ABB RAPID module: zignalmeister_2000.mod

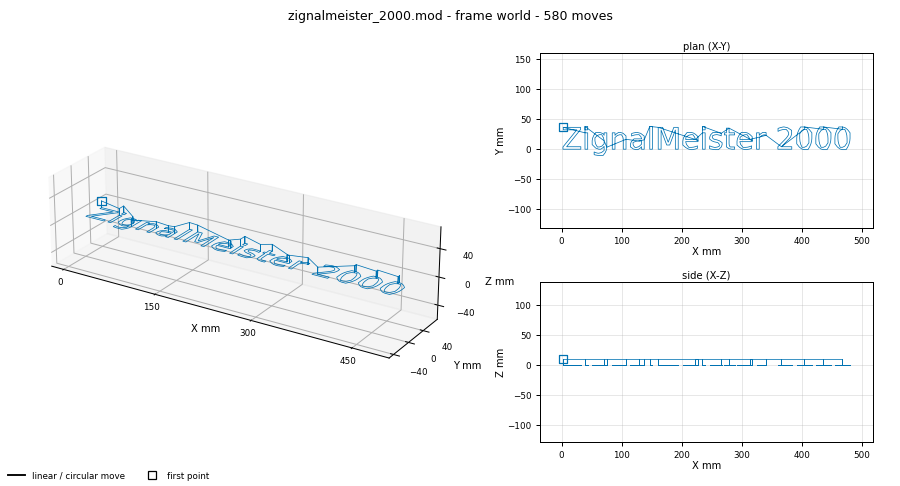
[picture p0: tool path of zignalmeister_2000.mod in frame world, 580 of 580 moves have a stored position in this frame; points joined in program order, loops and branches not executed]
MODULE TextDrawing
    ! Generated RAPID code for drawing text: ZignalMeister 2000
    ! Font: DejaVuSans.ttf
    ! Text size: 50.0 mm
    ! Point density: 5.0 mm
    ! Total points: 528
    ! Estimated time: 79.2 seconds

    ! Define target positions
    ! Path 1/26
    CONST robtarget p0:=[[2.81,36.45,0],[0,0,1,0],[-1,0,-1,0],[9E9,9E9,9E9,9E9,9E9,9E9]];
    CONST robtarget p1:=[[31.45,36.45,0],[0,0,1,0],[-1,0,-1,0],[9E9,9E9,9E9,9E9,9E9,9E9]];
    CONST robtarget p2:=[[31.45,32.69,0],[0,0,1,0],[-1,0,-1,0],[9E9,9E9,9E9,9E9,9E9,9E9]];
    CONST robtarget p3:=[[8.40,4.15,0],[0,0,1,0],[-1,0,-1,0],[9E9,9E9,9E9,9E9,9E9,9E9]];
    CONST robtarget p4:=[[32.01,4.15,0],[0,0,1,0],[-1,0,-1,0],[9E9,9E9,9E9,9E9,9E9,9E9]];
    CONST robtarget p5:=[[32.01,0.00,0],[0,0,1,0],[-1,0,-1,0],[9E9,9E9,9E9,9E9,9E9,9E9]];
    CONST robtarget p6:=[[2.25,0.00,0],[0,0,1,0],[-1,0,-1,0],[9E9,9E9,9E9,9E9,9E9,9E9]];
    CONST robtarget p7:=[[2.25,3.76,0],[0,0,1,0],[-1,0,-1,0],[9E9,9E9,9E9,9E9,9E9,9E9]];
    CONST robtarget p8:=[[25.29,32.30,0],[0,0,1,0],[-1,0,-1,0],[9E9,9E9,9E9,9E9,9E9,9E9]];
    CONST robtarget p9:=[[2.81,32.30,0],[0,0,1,0],[-1,0,-1,0],[9E9,9E9,9E9,9E9,9E9,9E9]];
    CONST robtarget p10:=[[2.81,36.45,0],[0,0,1,0],[-1,0,-1,0],[9E9,9E9,9E9,9E9,9E9,9E9]];
    ! Path 2/26
    CONST robtarget p11:=[[38.96,27.34,0],[0,0,1,0],[-1,0,-1,0],[9E9,9E9,9E9,9E9,9E9,9E9]];
    CONST robtarget p12:=[[43.46,27.34,0],[0,0,1,0],[-1,0,-1,0],[9E9,9E9,9E9,9E9,9E9,9E9]];
    CONST robtarget p13:=[[43.46,0.00,0],[0,0,1,0],[-1,0,-1,0],[9E9,9E9,9E9,9E9,9E9,9E9]];
    CONST robtarget p14:=[[38.96,0.00,0],[0,0,1,0],[-1,0,-1,0],[9E9,9E9,9E9,9E9,9E9,9E9]];
    CONST robtarget p15:=[[38.96,27.34,0],[0,0,1,0],[-1,0,-1,0],[9E9,9E9,9E9,9E9,9E9,9E9]];
    ! Path 3/26
    CONST robtarget p16:=[[38.96,37.99,0],[0,0,1,0],[-1,0,-1,0],[9E9,9E9,9E9,9E9,9E9,9E9]];
    CONST robtarget p17:=[[43.46,37.99,0],[0,0,1,0],[-1,0,-1,0],[9E9,9E9,9E9,9E9,9E9,9E9]];
    CONST robtarget p18:=[[43.46,32.30,0],[0,0,1,0],[-1,0,-1,0],[9E9,9E9,9E9,9E9,9E9,9E9]];
    CONST robtarget p19:=[[38.96,32.30,0],[0,0,1,0],[-1,0,-1,0],[9E9,9E9,9E9,9E9,9E9,9E9]];
    CONST robtarget p20:=[[38.96,37.99,0],[0,0,1,0],[-1,0,-1,0],[9E9,9E9,9E9,9E9,9E9,9E9]];
    ! Path 4/26
    CONST robtarget p21:=[[70.85,13.99,0],[0,0,1,0],[-1,0,-1,0],[9E9,9E9,9E9,9E9,9E9,9E9]];
    CONST robtarget p22:=[[69.84,18.99,0],[0,0,1,0],[-1,0,-1,0],[9E9,9E9,9E9,9E9,9E9,9E9]];
    CONST robtarget p23:=[[66.82,24.24,0],[0,0,1,0],[-1,0,-1,0],[9E9,9E9,9E9,9E9,9E9,9E9]];
    CONST robtarget p24:=[[65.91,24.24,0],[0,0,1,0],[-1,0,-1,0],[9E9,9E9,9E9,9E9,9E9,9E9]];
    CONST robtarget p25:=[[63.18,24.24,0],[0,0,1,0],[-1,0,-1,0],[9E9,9E9,9E9,9E9,9E9,9E9]];
    CONST robtarget p26:=[[59.47,22.90,0],[0,0,1,0],[-1,0,-1,0],[9E9,9E9,9E9,9E9,9E9,9E9]];
    CONST robtarget p27:=[[55.54,18.87,0],[0,0,1,0],[-1,0,-1,0],[9E9,9E9,9E9,9E9,9E9,9E9]];
    CONST robtarget p28:=[[55.54,17.65,0],[0,0,1,0],[-1,0,-1,0],[9E9,9E9,9E9,9E9,9E9,9E9]];
    CONST robtarget p29:=[[55.54,13.99,0],[0,0,1,0],[-1,0,-1,0],[9E9,9E9,9E9,9E9,9E9,9E9]];
    CONST robtarget p30:=[[56.55,9.00,0],[0,0,1,0],[-1,0,-1,0],[9E9,9E9,9E9,9E9,9E9,9E9]];
    CONST robtarget p31:=[[59.57,3.76,0],[0,0,1,0],[-1,0,-1,0],[9E9,9E9,9E9,9E9,9E9,9E9]];
    CONST robtarget p32:=[[60.47,3.76,0],[0,0,1,0],[-1,0,-1,0],[9E9,9E9,9E9,9E9,9E9,9E9]];
    CONST robtarget p33:=[[63.18,3.76,0],[0,0,1,0],[-1,0,-1,0],[9E9,9E9,9E9,9E9,9E9,9E9]];
    CONST robtarget p34:=[[66.92,5.10,0],[0,0,1,0],[-1,0,-1,0],[9E9,9E9,9E9,9E9,9E9,9E9]];
    CONST robtarget p35:=[[70.85,9.13,0],[0,0,1,0],[-1,0,-1,0],[9E9,9E9,9E9,9E9,9E9,9E9]];
    CONST robtarget p36:=[[70.85,10.35,0],[0,0,1,0],[-1,0,-1,0],[9E9,9E9,9E9,9E9,9E9,9E9]];
    CONST robtarget p37:=[[70.85,13.99,0],[0,0,1,0],[-1,0,-1,0],[9E9,9E9,9E9,9E9,9E9,9E9]];
    ! Path 5/26
    CONST robtarget p38:=[[75.34,3.39,0],[0,0,1,0],[-1,0,-1,0],[9E9,9E9,9E9,9E9,9E9,9E9]];
    CONST robtarget p39:=[[74.65,-1.24,0],[0,0,1,0],[-1,0,-1,0],[9E9,9E9,9E9,9E9,9E9,9E9]];
    CONST robtarget p40:=[[72.59,-5.84,0],[0,0,1,0],[-1,0,-1,0],[9E9,9E9,9E9,9E9,9E9,9E9]];
    CONST robtarget p41:=[[69.14,-10.40,0],[0,0,1,0],[-1,0,-1,0],[9E9,9E9,9E9,9E9,9E9,9E9]];
    CONST robtarget p42:=[[67.54,-10.40,0],[0,0,1,0],[-1,0,-1,0],[9E9,9E9,9E9,9E9,9E9,9E9]];
    CONST robtarget p43:=[[62.74,-10.40,0],[0,0,1,0],[-1,0,-1,0],[9E9,9E9,9E9,9E9,9E9,9E9]];
    CONST robtarget p44:=[[59.92,-10.22,0],[0,0,1,0],[-1,0,-1,0],[9E9,9E9,9E9,9E9,9E9,9E9]];
    CONST robtarget p45:=[[56.18,-9.69,0],[0,0,1,0],[-1,0,-1,0],[9E9,9E9,9E9,9E9,9E9,9E9]];
    CONST robtarget p46:=[[55.68,-9.51,0],[0,0,1,0],[-1,0,-1,0],[9E9,9E9,9E9,9E9,9E9,9E9]];
    CONST robtarget p47:=[[54.20,-8.96,0],[0,0,1,0],[-1,0,-1,0],[9E9,9E9,9E9,9E9,9E9,9E9]];
    CONST robtarget p48:=[[54.20,-4.59,0],[0,0,1,0],[-1,0,-1,0],[9E9,9E9,9E9,9E9,9E9,9E9]];
    CONST robtarget p49:=[[56.65,-5.65,0],[0,0,1,0],[-1,0,-1,0],[9E9,9E9,9E9,9E9,9E9,9E9]];
    CONST robtarget p50:=[[60.03,-6.69,0],[0,0,1,0],[-1,0,-1,0],[9E9,9E9,9E9,9E9,9E9,9E9]];
    CONST robtarget p51:=[[60.53,-6.69,0],[0,0,1,0],[-1,0,-1,0],[9E9,9E9,9E9,9E9,9E9,9E9]];
    CONST robtarget p52:=[[62.04,-6.69,0],[0,0,1,0],[-1,0,-1,0],[9E9,9E9,9E9,9E9,9E9,9E9]];
    CONST robtarget p53:=[[66.45,-5.54,0],[0,0,1,0],[-1,0,-1,0],[9E9,9E9,9E9,9E9,9E9,9E9]];
    CONST robtarget p54:=[[70.85,-2.08,0],[0,0,1,0],[-1,0,-1,0],[9E9,9E9,9E9,9E9,9E9,9E9]];
    CONST robtarget p55:=[[70.85,-0.91,0],[0,0,1,0],[-1,0,-1,0],[9E9,9E9,9E9,9E9,9E9,9E9]];
    CONST robtarget p56:=[[70.85,2.59,0],[0,0,1,0],[-1,0,-1,0],[9E9,9E9,9E9,9E9,9E9,9E9]];
    CONST robtarget p57:=[[70.85,4.81,0],[0,0,1,0],[-1,0,-1,0],[9E9,9E9,9E9,9E9,9E9,9E9]];
    CONST robtarget p58:=[[68.72,2.40,0],[0,0,1,0],[-1,0,-1,0],[9E9,9E9,9E9,9E9,9E9,9E9]];
    CONST robtarget p59:=[[65.11,0.00,0],[0,0,1,0],[-1,0,-1,0],[9E9,9E9,9E9,9E9,9E9,9E9]];
    CONST robtarget p60:=[[64.36,0.00,0],[0,0,1,0],[-1,0,-1,0],[9E9,9E9,9E9,9E9,9E9,9E9]];
    CONST robtarget p61:=[[62.08,0.00,0],[0,0,1,0],[-1,0,-1,0],[9E9,9E9,9E9,9E9,9E9,9E9]];
    CONST robtarget p62:=[[56.77,1.92,0],[0,0,1,0],[-1,0,-1,0],[9E9,9E9,9E9,9E9,9E9,9E9]];
    CONST robtarget p63:=[[50.90,7.67,0],[0,0,1,0],[-1,0,-1,0],[9E9,9E9,9E9,9E9,9E9,9E9]];
    CONST robtarget p64:=[[50.90,9.25,0],[0,0,1,0],[-1,0,-1,0],[9E9,9E9,9E9,9E9,9E9,9E9]];
    CONST robtarget p65:=[[50.90,13.99,0],[0,0,1,0],[-1,0,-1,0],[9E9,9E9,9E9,9E9,9E9,9E9]];
    CONST robtarget p66:=[[51.59,18.37,0],[0,0,1,0],[-1,0,-1,0],[9E9,9E9,9E9,9E9,9E9,9E9]];
    CONST robtarget p67:=[[53.64,23.04,0],[0,0,1,0],[-1,0,-1,0],[9E9,9E9,9E9,9E9,9E9,9E9]];
    CONST robtarget p68:=[[57.06,28.00,0],[0,0,1,0],[-1,0,-1,0],[9E9,9E9,9E9,9E9,9E9,9E9]];
    CONST robtarget p69:=[[58.31,28.00,0],[0,0,1,0],[-1,0,-1,0],[9E9,9E9,9E9,9E9,9E9,9E9]];
    CONST robtarget p70:=[[62.08,28.00,0],[0,0,1,0],[-1,0,-1,0],[9E9,9E9,9E9,9E9,9E9,9E9]];
    CONST robtarget p71:=[[65.44,27.40,0],[0,0,1,0],[-1,0,-1,0],[9E9,9E9,9E9,9E9,9E9,9E9]];
    CONST robtarget p72:=[[69.46,25.61,0],[0,0,1,0],[-1,0,-1,0],[9E9,9E9,9E9,9E9,9E9,9E9]];
    CONST robtarget p73:=[[69.81,25.01,0],[0,0,1,0],[-1,0,-1,0],[9E9,9E9,9E9,9E9,9E9,9E9]];
    CONST robtarget p74:=[[70.85,23.19,0],[0,0,1,0],[-1,0,-1,0],[9E9,9E9,9E9,9E9,9E9,9E9]];
    CONST robtarget p75:=[[70.85,27.34,0],[0,0,1,0],[-1,0,-1,0],[9E9,9E9,9E9,9E9,9E9,9E9]];
    CONST robtarget p76:=[[75.34,27.34,0],[0,0,1,0],[-1,0,-1,0],[9E9,9E9,9E9,9E9,9E9,9E9]];
    CONST robtarget p77:=[[75.34,3.39,0],[0,0,1,0],[-1,0,-1,0],[9E9,9E9,9E9,9E9,9E9,9E9]];
    ! Path 6/26
    CONST robtarget p78:=[[107.32,16.50,0],[0,0,1,0],[-1,0,-1,0],[9E9,9E9,9E9,9E9,9E9,9E9]];
    CONST robtarget p79:=[[107.32,0.00,0],[0,0,1,0],[-1,0,-1,0],[9E9,9E9,9E9,9E9,9E9,9E9]];
    CONST robtarget p80:=[[102.83,0.00,0],[0,0,1,0],[-1,0,-1,0],[9E9,9E9,9E9,9E9,9E9,9E9]];
    CONST robtarget p81:=[[102.83,16.36,0],[0,0,1,0],[-1,0,-1,0],[9E9,9E9,9E9,9E9,9E9,9E9]];
    CONST robtarget p82:=[[102.08,20.23,0],[0,0,1,0],[-1,0,-1,0],[9E9,9E9,9E9,9E9,9E9,9E9]];
    CONST robtarget p83:=[[99.80,24.10,0],[0,0,1,0],[-1,0,-1,0],[9E9,9E9,9E9,9E9,9E9,9E9]];
    CONST robtarget p84:=[[99.05,24.10,0],[0,0,1,0],[-1,0,-1,0],[9E9,9E9,9E9,9E9,9E9,9E9]];
    CONST robtarget p85:=[[96.78,24.10,0],[0,0,1,0],[-1,0,-1,0],[9E9,9E9,9E9,9E9,9E9,9E9]];
    CONST robtarget p86:=[[93.00,22.94,0],[0,0,1,0],[-1,0,-1,0],[9E9,9E9,9E9,9E9,9E9,9E9]];
    CONST robtarget p87:=[[88.94,19.46,0],[0,0,1,0],[-1,0,-1,0],[9E9,9E9,9E9,9E9,9E9,9E9]];
    CONST robtarget p88:=[[88.94,18.46,0],[0,0,1,0],[-1,0,-1,0],[9E9,9E9,9E9,9E9,9E9,9E9]];
    CONST robtarget p89:=[[88.94,15.45,0],[0,0,1,0],[-1,0,-1,0],[9E9,9E9,9E9,9E9,9E9,9E9]];
    CONST robtarget p90:=[[88.94,0.00,0],[0,0,1,0],[-1,0,-1,0],[9E9,9E9,9E9,9E9,9E9,9E9]];
    CONST robtarget p91:=[[84.42,0.00,0],[0,0,1,0],[-1,0,-1,0],[9E9,9E9,9E9,9E9,9E9,9E9]];
    CONST robtarget p92:=[[84.42,27.34,0],[0,0,1,0],[-1,0,-1,0],[9E9,9E9,9E9,9E9,9E9,9E9]];
    CONST robtarget p93:=[[88.94,27.34,0],[0,0,1,0],[-1,0,-1,0],[9E9,9E9,9E9,9E9,9E9,9E9]];
    CONST robtarget p94:=[[88.94,23.10,0],[0,0,1,0],[-1,0,-1,0],[9E9,9E9,9E9,9E9,9E9,9E9]];
    CONST robtarget p95:=[[91.24,25.56,0],[0,0,1,0],[-1,0,-1,0],[9E9,9E9,9E9,9E9,9E9,9E9]];
    CONST robtarget p96:=[[94.92,28.00,0],[0,0,1,0],[-1,0,-1,0],[9E9,9E9,9E9,9E9,9E9,9E9]];
    CONST robtarget p97:=[[95.64,28.00,0],[0,0,1,0],[-1,0,-1,0],[9E9,9E9,9E9,9E9,9E9,9E9]];
    CONST robtarget p98:=[[97.78,28.00,0],[0,0,1,0],[-1,0,-1,0],[9E9,9E9,9E9,9E9,9E9,9E9]];
    CONST robtarget p99:=[[102.52,26.54,0],[0,0,1,0],[-1,0,-1,0],[9E9,9E9,9E9,9E9,9E9,9E9]];
    CONST robtarget p100:=[[107.32,22.17,0],[0,0,1,0],[-1,0,-1,0],[9E9,9E9,9E9,9E9,9E9,9E9]];
    CONST robtarget p101:=[[107.32,20.75,0],[0,0,1,0],[-1,0,-1,0],[9E9,9E9,9E9,9E9,9E9,9E9]];
    CONST robtarget p102:=[[107.32,16.50,0],[0,0,1,0],[-1,0,-1,0],[9E9,9E9,9E9,9E9,9E9,9E9]];
    ! Path 7/26
    CONST robtarget p103:=[[128.71,13.75,0],[0,0,1,0],[-1,0,-1,0],[9E9,9E9,9E9,9E9,9E9,9E9]];
    CONST robtarget p104:=[[123.58,13.12,0],[0,0,1,0],[-1,0,-1,0],[9E9,9E9,9E9,9E9,9E9,9E9]];
    CONST robtarget p105:=[[119.07,11.25,0],[0,0,1,0],[-1,0,-1,0],[9E9,9E9,9E9,9E9,9E9,9E9]];
    CONST robtarget p106:=[[119.07,10.50,0],[0,0,1,0],[-1,0,-1,0],[9E9,9E9,9E9,9E9,9E9,9E9]];
    CONST robtarget p107:=[[119.07,8.25,0],[0,0,1,0],[-1,0,-1,0],[9E9,9E9,9E9,9E9,9E9,9E9]];
    CONST robtarget p108:=[[119.85,5.76,0],[0,0,1,0],[-1,0,-1,0],[9E9,9E9,9E9,9E9,9E9,9E9]];
    CONST robtarget p109:=[[122.22,3.05,0],[0,0,1,0],[-1,0,-1,0],[9E9,9E9,9E9,9E9,9E9,9E9]];
    CONST robtarget p110:=[[122.89,3.05,0],[0,0,1,0],[-1,0,-1,0],[9E9,9E9,9E9,9E9,9E9,9E9]];
    CONST robtarget p111:=[[124.93,3.05,0],[0,0,1,0],[-1,0,-1,0],[9E9,9E9,9E9,9E9,9E9,9E9]];
    CONST robtarget p112:=[[128.86,4.38,0],[0,0,1,0],[-1,0,-1,0],[9E9,9E9,9E9,9E9,9E9,9E9]];
    CONST robtarget p113:=[[133.18,8.35,0],[0,0,1,0],[-1,0,-1,0],[9E9,9E9,9E9,9E9,9E9,9E9]];
    CONST robtarget p114:=[[133.18,9.45,0],[0,0,1,0],[-1,0,-1,0],[9E9,9E9,9E9,9E9,9E9,9E9]];
    CONST robtarget p115:=[[133.18,12.74,0],[0,0,1,0],[-1,0,-1,0],[9E9,9E9,9E9,9E9,9E9,9E9]];
    CONST robtarget p116:=[[133.18,13.75,0],[0,0,1,0],[-1,0,-1,0],[9E9,9E9,9E9,9E9,9E9,9E9]];
    CONST robtarget p117:=[[128.71,13.75,0],[0,0,1,0],[-1,0,-1,0],[9E9,9E9,9E9,9E9,9E9,9E9]];
    ! Path 8/26
    CONST robtarget p118:=[[137.67,15.60,0],[0,0,1,0],[-1,0,-1,0],[9E9,9E9,9E9,9E9,9E9,9E9]];
    CONST robtarget p119:=[[137.67,0.00,0],[0,0,1,0],[-1,0,-1,0],[9E9,9E9,9E9,9E9,9E9,9E9]];
    CONST robtarget p120:=[[133.18,0.00,0],[0,0,1,0],[-1,0,-1,0],[9E9,9E9,9E9,9E9,9E9,9E9]];
    CONST robtarget p121:=[[133.18,4.15,0],[0,0,1,0],[-1,0,-1,0],[9E9,9E9,9E9,9E9,9E9,9E9]];
    CONST robtarget p122:=[[130.88,1.69,0],[0,0,1,0],[-1,0,-1,0],[9E9,9E9,9E9,9E9,9E9,9E9]];
    CONST robtarget p123:=[[127.05,-0.71,0],[0,0,1,0],[-1,0,-1,0],[9E9,9E9,9E9,9E9,9E9,9E9]];
    CONST robtarget p124:=[[126.22,-0.71,0],[0,0,1,0],[-1,0,-1,0],[9E9,9E9,9E9,9E9,9E9,9E9]];
    CONST robtarget p125:=[[123.73,-0.71,0],[0,0,1,0],[-1,0,-1,0],[9E9,9E9,9E9,9E9,9E9,9E9]];
    CONST robtarget p126:=[[119.34,0.47,0],[0,0,1,0],[-1,0,-1,0],[9E9,9E9,9E9,9E9,9E9,9E9]];
    CONST robtarget p127:=[[114.58,4.00,0],[0,0,1,0],[-1,0,-1,0],[9E9,9E9,9E9,9E9,9E9,9E9]];
    CONST robtarget p128:=[[114.58,4.99,0],[0,0,1,0],[-1,0,-1,0],[9E9,9E9,9E9,9E9,9E9,9E9]];
    CONST robtarget p129:=[[114.58,7.96,0],[0,0,1,0],[-1,0,-1,0],[9E9,9E9,9E9,9E9,9E9,9E9]];
    CONST robtarget p130:=[[116.12,12.59,0],[0,0,1,0],[-1,0,-1,0],[9E9,9E9,9E9,9E9,9E9,9E9]];
    CONST robtarget p131:=[[120.75,17.26,0],[0,0,1,0],[-1,0,-1,0],[9E9,9E9,9E9,9E9,9E9,9E9]];
    CONST robtarget p132:=[[122.28,17.26,0],[0,0,1,0],[-1,0,-1,0],[9E9,9E9,9E9,9E9,9E9,9E9]];
    CONST robtarget p133:=[[126.88,17.26,0],[0,0,1,0],[-1,0,-1,0],[9E9,9E9,9E9,9E9,9E9,9E9]];
    CONST robtarget p134:=[[133.18,17.26,0],[0,0,1,0],[-1,0,-1,0],[9E9,9E9,9E9,9E9,9E9,9E9]];
    CONST robtarget p135:=[[133.18,17.70,0],[0,0,1,0],[-1,0,-1,0],[9E9,9E9,9E9,9E9,9E9,9E9]];
    CONST robtarget p136:=[[132.16,20.87,0],[0,0,1,0],[-1,0,-1,0],[9E9,9E9,9E9,9E9,9E9,9E9]];
    CONST robtarget p137:=[[129.10,24.19,0],[0,0,1,0],[-1,0,-1,0],[9E9,9E9,9E9,9E9,9E9,9E9]];
    CONST robtarget p138:=[[128.18,24.19,0],[0,0,1,0],[-1,0,-1,0],[9E9,9E9,9E9,9E9,9E9,9E9]];
    CONST robtarget p139:=[[125.42,24.19,0],[0,0,1,0],[-1,0,-1,0],[9E9,9E9,9E9,9E9,9E9,9E9]];
    CONST robtarget p140:=[[122.55,23.91,0],[0,0,1,0],[-1,0,-1,0],[9E9,9E9,9E9,9E9,9E9,9E9]];
    CONST robtarget p141:=[[118.63,23.07,0],[0,0,1,0],[-1,0,-1,0],[9E9,9E9,9E9,9E9,9E9,9E9]];
    CONST robtarget p142:=[[118.12,22.79,0],[0,0,1,0],[-1,0,-1,0],[9E9,9E9,9E9,9E9,9E9,9E9]];
    CONST robtarget p143:=[[116.58,21.95,0],[0,0,1,0],[-1,0,-1,0],[9E9,9E9,9E9,9E9,9E9,9E9]];
    CONST robtarget p144:=[[116.58,26.10,0],[0,0,1,0],[-1,0,-1,0],[9E9,9E9,9E9,9E9,9E9,9E9]];
    CONST robtarget p145:=[[119.59,27.05,0],[0,0,1,0],[-1,0,-1,0],[9E9,9E9,9E9,9E9,9E9,9E9]];
    CONST robtarget p146:=[[123.68,28.00,0],[0,0,1,0],[-1,0,-1,0],[9E9,9E9,9E9,9E9,9E9,9E9]];
    CONST robtarget p147:=[[124.23,28.00,0],[0,0,1,0],[-1,0,-1,0],[9E9,9E9,9E9,9E9,9E9,9E9]];
    CONST robtarget p148:=[[125.88,28.00,0],[0,0,1,0],[-1,0,-1,0],[9E9,9E9,9E9,9E9,9E9,9E9]];
    CONST robtarget p149:=[[131.79,26.46,0],[0,0,1,0],[-1,0,-1,0],[9E9,9E9,9E9,9E9,9E9,9E9]];
    CONST robtarget p150:=[[137.67,21.85,0],[0,0,1,0],[-1,0,-1,0],[9E9,9E9,9E9,9E9,9E9,9E9]];
    CONST robtarget p151:=[[137.67,20.29,0],[0,0,1,0],[-1,0,-1,0],[9E9,9E9,9E9,9E9,9E9,9E9]];
    CONST robtarget p152:=[[137.67,15.60,0],[0,0,1,0],[-1,0,-1,0],[9E9,9E9,9E9,9E9,9E9,9E9]];
    ! Path 9/26
    CONST robtarget p153:=[[146.92,37.99,0],[0,0,1,0],[-1,0,-1,0],[9E9,9E9,9E9,9E9,9E9,9E9]];
    CONST robtarget p154:=[[151.42,37.99,0],[0,0,1,0],[-1,0,-1,0],[9E9,9E9,9E9,9E9,9E9,9E9]];
    CONST robtarget p155:=[[151.42,0.00,0],[0,0,1,0],[-1,0,-1,0],[9E9,9E9,9E9,9E9,9E9,9E9]];
    CONST robtarget p156:=[[146.92,0.00,0],[0,0,1,0],[-1,0,-1,0],[9E9,9E9,9E9,9E9,9E9,9E9]];
    CONST robtarget p157:=[[146.92,37.99,0],[0,0,1,0],[-1,0,-1,0],[9E9,9E9,9E9,9E9,9E9,9E9]];
    ! Path 10/26
    CONST robtarget p158:=[[161.01,36.45,0],[0,0,1,0],[-1,0,-1,0],[9E9,9E9,9E9,9E9,9E9,9E9]];
    CONST robtarget p159:=[[168.36,36.45,0],[0,0,1,0],[-1,0,-1,0],[9E9,9E9,9E9,9E9,9E9,9E9]];
    CONST robtarget p160:=[[177.66,11.65,0],[0,0,1,0],[-1,0,-1,0],[9E9,9E9,9E9,9E9,9E9,9E9]];
    CONST robtarget p161:=[[187.01,36.45,0],[0,0,1,0],[-1,0,-1,0],[9E9,9E9,9E9,9E9,9E9,9E9]];
    CONST robtarget p162:=[[194.36,36.45,0],[0,0,1,0],[-1,0,-1,0],[9E9,9E9,9E9,9E9,9E9,9E9]];
    CONST robtarget p163:=[[194.36,0.00,0],[0,0,1,0],[-1,0,-1,0],[9E9,9E9,9E9,9E9,9E9,9E9]];
    CONST robtarget p164:=[[189.55,0.00,0],[0,0,1,0],[-1,0,-1,0],[9E9,9E9,9E9,9E9,9E9,9E9]];
    CONST robtarget p165:=[[189.55,32.01,0],[0,0,1,0],[-1,0,-1,0],[9E9,9E9,9E9,9E9,9E9,9E9]];
    CONST robtarget p166:=[[180.15,7.01,0],[0,0,1,0],[-1,0,-1,0],[9E9,9E9,9E9,9E9,9E9,9E9]];
    CONST robtarget p167:=[[175.20,7.01,0],[0,0,1,0],[-1,0,-1,0],[9E9,9E9,9E9,9E9,9E9,9E9]];
    CONST robtarget p168:=[[165.80,32.01,0],[0,0,1,0],[-1,0,-1,0],[9E9,9E9,9E9,9E9,9E9,9E9]];
    CONST robtarget p169:=[[165.80,0.00,0],[0,0,1,0],[-1,0,-1,0],[9E9,9E9,9E9,9E9,9E9,9E9]];
    CONST robtarget p170:=[[161.01,0.00,0],[0,0,1,0],[-1,0,-1,0],[9E9,9E9,9E9,9E9,9E9,9E9]];
    CONST robtarget p171:=[[161.01,36.45,0],[0,0,1,0],[-1,0,-1,0],[9E9,9E9,9E9,9E9,9E9,9E9]];
    ! Path 11/26
    CONST robtarget p172:=[[227.34,14.79,0],[0,0,1,0],[-1,0,-1,0],[9E9,9E9,9E9,9E9,9E9,9E9]];
    CONST robtarget p173:=[[227.34,12.60,0],[0,0,1,0],[-1,0,-1,0],[9E9,9E9,9E9,9E9,9E9,9E9]];
    CONST robtarget p174:=[[206.69,12.60,0],[0,0,1,0],[-1,0,-1,0],[9E9,9E9,9E9,9E9,9E9,9E9]];
    CONST robtarget p175:=[[208.16,7.90,0],[0,0,1,0],[-1,0,-1,0],[9E9,9E9,9E9,9E9,9E9,9E9]];
    CONST robtarget p176:=[[211.99,3.10,0],[0,0,1,0],[-1,0,-1,0],[9E9,9E9,9E9,9E9,9E9,9E9]];
    CONST robtarget p177:=[[213.10,3.10,0],[0,0,1,0],[-1,0,-1,0],[9E9,9E9,9E9,9E9,9E9,9E9]];
    CONST robtarget p178:=[[216.46,3.10,0],[0,0,1,0],[-1,0,-1,0],[9E9,9E9,9E9,9E9,9E9,9E9]];
    CONST robtarget p179:=[[219.61,3.42,0],[0,0,1,0],[-1,0,-1,0],[9E9,9E9,9E9,9E9,9E9,9E9]];
    CONST robtarget p180:=[[223.90,4.37,0],[0,0,1,0],[-1,0,-1,0],[9E9,9E9,9E9,9E9,9E9,9E9]];
    CONST robtarget p181:=[[224.50,4.69,0],[0,0,1,0],[-1,0,-1,0],[9E9,9E9,9E9,9E9,9E9,9E9]];
    CONST robtarget p182:=[[226.29,5.64,0],[0,0,1,0],[-1,0,-1,0],[9E9,9E9,9E9,9E9,9E9,9E9]];
    CONST robtarget p183:=[[226.29,1.39,0],[0,0,1,0],[-1,0,-1,0],[9E9,9E9,9E9,9E9,9E9,9E9]];
    CONST robtarget p184:=[[223.21,0.35,0],[0,0,1,0],[-1,0,-1,0],[9E9,9E9,9E9,9E9,9E9,9E9]];
    CONST robtarget p185:=[[218.80,-0.71,0],[0,0,1,0],[-1,0,-1,0],[9E9,9E9,9E9,9E9,9E9,9E9]];
    CONST robtarget p186:=[[218.15,-0.71,0],[0,0,1,0],[-1,0,-1,0],[9E9,9E9,9E9,9E9,9E9,9E9]];
    CONST robtarget p187:=[[216.19,-0.71,0],[0,0,1,0],[-1,0,-1,0],[9E9,9E9,9E9,9E9,9E9,9E9]];
    CONST robtarget p188:=[[211.70,0.14,0],[0,0,1,0],[-1,0,-1,0],[9E9,9E9,9E9,9E9,9E9,9E9]];
    CONST robtarget p189:=[[206.97,2.68,0],[0,0,1,0],[-1,0,-1,0],[9E9,9E9,9E9,9E9,9E9,9E9]];
    CONST robtarget p190:=[[202.00,6.91,0],[0,0,1,0],[-1,0,-1,0],[9E9,9E9,9E9,9E9,9E9,9E9]];
    CONST robtarget p191:=[[202.00,8.53,0],[0,0,1,0],[-1,0,-1,0],[9E9,9E9,9E9,9E9,9E9,9E9]];
    CONST robtarget p192:=[[202.00,13.40,0],[0,0,1,0],[-1,0,-1,0],[9E9,9E9,9E9,9E9,9E9,9E9]];
    CONST robtarget p193:=[[202.81,18.01,0],[0,0,1,0],[-1,0,-1,0],[9E9,9E9,9E9,9E9,9E9,9E9]];
    CONST robtarget p194:=[[205.22,22.88,0],[0,0,1,0],[-1,0,-1,0],[9E9,9E9,9E9,9E9,9E9,9E9]];
    CONST robtarget p195:=[[209.25,28.00,0],[0,0,1,0],[-1,0,-1,0],[9E9,9E9,9E9,9E9,9E9,9E9]];
    CONST robtarget p196:=[[210.79,28.00,0],[0,0,1,0],[-1,0,-1,0],[9E9,9E9,9E9,9E9,9E9,9E9]];
    CONST robtarget p197:=[[215.41,28.00,0],[0,0,1,0],[-1,0,-1,0],[9E9,9E9,9E9,9E9,9E9,9E9]];
    CONST robtarget p198:=[[219.18,27.21,0],[0,0,1,0],[-1,0,-1,0],[9E9,9E9,9E9,9E9,9E9,9E9]];
    CONST robtarget p199:=[[223.16,24.85,0],[0,0,1,0],[-1,0,-1,0],[9E9,9E9,9E9,9E9,9E9,9E9]];
    CONST robtarget p200:=[[227.34,20.90,0],[0,0,1,0],[-1,0,-1,0],[9E9,9E9,9E9,9E9,9E9,9E9]];
    CONST robtarget p201:=[[227.34,19.37,0],[0,0,1,0],[-1,0,-1,0],[9E9,9E9,9E9,9E9,9E9,9E9]];
    CONST robtarget p202:=[[227.34,14.79,0],[0,0,1,0],[-1,0,-1,0],[9E9,9E9,9E9,9E9,9E9,9E9]];
    ! Path 12/26
    CONST robtarget p203:=[[222.85,16.11,0],[0,0,1,0],[-1,0,-1,0],[9E9,9E9,9E9,9E9,9E9,9E9]];
    CONST robtarget p204:=[[221.81,19.98,0],[0,0,1,0],[-1,0,-1,0],[9E9,9E9,9E9,9E9,9E9,9E9]];
    CONST robtarget p205:=[[218.77,24.19,0],[0,0,1,0],[-1,0,-1,0],[9E9,9E9,9E9,9E9,9E9,9E9]];
    CONST robtarget p206:=[[217.94,24.19,0],[0,0,1,0],[-1,0,-1,0],[9E9,9E9,9E9,9E9,9E9,9E9]];
    CONST robtarget p207:=[[215.45,24.19,0],[0,0,1,0],[-1,0,-1,0],[9E9,9E9,9E9,9E9,9E9,9E9]];
    CONST robtarget p208:=[[211.51,23.13,0],[0,0,1,0],[-1,0,-1,0],[9E9,9E9,9E9,9E9,9E9,9E9]];
    CONST robtarget p209:=[[207.18,19.95,0],[0,0,1,0],[-1,0,-1,0],[9E9,9E9,9E9,9E9,9E9,9E9]];
    CONST robtarget p210:=[[207.09,18.98,0],[0,0,1,0],[-1,0,-1,0],[9E9,9E9,9E9,9E9,9E9,9E9]];
    CONST robtarget p211:=[[206.84,16.09,0],[0,0,1,0],[-1,0,-1,0],[9E9,9E9,9E9,9E9,9E9,9E9]];
    CONST robtarget p212:=[[222.85,16.11,0],[0,0,1,0],[-1,0,-1,0],[9E9,9E9,9E9,9E9,9E9,9E9]];
    ! Path 13/26
    CONST robtarget p213:=[[234.72,27.34,0],[0,0,1,0],[-1,0,-1,0],[9E9,9E9,9E9,9E9,9E9,9E9]];
    CONST robtarget p214:=[[239.21,27.34,0],[0,0,1,0],[-1,0,-1,0],[9E9,9E9,9E9,9E9,9E9,9E9]];
    CONST robtarget p215:=[[239.21,0.00,0],[0,0,1,0],[-1,0,-1,0],[9E9,9E9,9E9,9E9,9E9,9E9]];
    CONST robtarget p216:=[[234.72,0.00,0],[0,0,1,0],[-1,0,-1,0],[9E9,9E9,9E9,9E9,9E9,9E9]];
    CONST robtarget p217:=[[234.72,27.34,0],[0,0,1,0],[-1,0,-1,0],[9E9,9E9,9E9,9E9,9E9,9E9]];
    ! Path 14/26
    CONST robtarget p218:=[[234.72,37.99,0],[0,0,1,0],[-1,0,-1,0],[9E9,9E9,9E9,9E9,9E9,9E9]];
    CONST robtarget p219:=[[239.21,37.99,0],[0,0,1,0],[-1,0,-1,0],[9E9,9E9,9E9,9E9,9E9,9E9]];
    CONST robtarget p220:=[[239.21,32.30,0],[0,0,1,0],[-1,0,-1,0],[9E9,9E9,9E9,9E9,9E9,9E9]];
    CONST robtarget p221:=[[234.72,32.30,0],[0,0,1,0],[-1,0,-1,0],[9E9,9E9,9E9,9E9,9E9,9E9]];
    CONST robtarget p222:=[[234.72,37.99,0],[0,0,1,0],[-1,0,-1,0],[9E9,9E9,9E9,9E9,9E9,9E9]];
    ! Path 15/26
    CONST robtarget p223:=[[266.04,26.54,0],[0,0,1,0],[-1,0,-1,0],[9E9,9E9,9E9,9E9,9E9,9E9]];
    CONST robtarget p224:=[[266.04,22.29,0],[0,0,1,0],[-1,0,-1,0],[9E9,9E9,9E9,9E9,9E9,9E9]];
    CONST robtarget p225:=[[263.59,23.27,0],[0,0,1,0],[-1,0,-1,0],[9E9,9E9,9E9,9E9,9E9,9E9]];
    CONST robtarget p226:=[[260.03,24.24,0],[0,0,1,0],[-1,0,-1,0],[9E9,9E9,9E9,9E9,9E9,9E9]];
    CONST robtarget p227:=[[259.48,24.24,0],[0,0,1,0],[-1,0,-1,0],[9E9,9E9,9E9,9E9,9E9,9E9]];
    CONST robtarget p228:=[[257.84,24.24,0],[0,0,1,0],[-1,0,-1,0],[9E9,9E9,9E9,9E9,9E9,9E9]];
    CONST robtarget p229:=[[254.49,23.73,0],[0,0,1,0],[-1,0,-1,0],[9E9,9E9,9E9,9E9,9E9,9E9]];
    CONST robtarget p230:=[[251.15,22.19,0],[0,0,1,0],[-1,0,-1,0],[9E9,9E9,9E9,9E9,9E9,9E9]];
    CONST robtarget p231:=[[251.15,21.68,0],[0,0,1,0],[-1,0,-1,0],[9E9,9E9,9E9,9E9,9E9,9E9]];
    CONST robtarget p232:=[[251.15,20.14,0],[0,0,1,0],[-1,0,-1,0],[9E9,9E9,9E9,9E9,9E9,9E9]];
    CONST robtarget p233:=[[251.75,18.52,0],[0,0,1,0],[-1,0,-1,0],[9E9,9E9,9E9,9E9,9E9,9E9]];
    CONST robtarget p234:=[[253.54,16.80,0],[0,0,1,0],[-1,0,-1,0],[9E9,9E9,9E9,9E9,9E9,9E9]];
    CONST robtarget p235:=[[254.44,16.60,0],[0,0,1,0],[-1,0,-1,0],[9E9,9E9,9E9,9E9,9E9,9E9]];
    CONST robtarget p236:=[[257.15,15.99,0],[0,0,1,0],[-1,0,-1,0],[9E9,9E9,9E9,9E9,9E9,9E9]];
    CONST robtarget p237:=[[258.69,15.65,0],[0,0,1,0],[-1,0,-1,0],[9E9,9E9,9E9,9E9,9E9,9E9]];
    CONST robtarget p238:=[[263.29,13.95,0],[0,0,1,0],[-1,0,-1,0],[9E9,9E9,9E9,9E9,9E9,9E9]];
    CONST robtarget p239:=[[267.50,10.89,0],[0,0,1,0],[-1,0,-1,0],[9E9,9E9,9E9,9E9,9E9,9E9]];
    CONST robtarget p240:=[[267.50,10.05,0],[0,0,1,0],[-1,0,-1,0],[9E9,9E9,9E9,9E9,9E9,9E9]];
    CONST robtarget p241:=[[267.50,7.54,0],[0,0,1,0],[-1,0,-1,0],[9E9,9E9,9E9,9E9,9E9,9E9]];
    CONST robtarget p242:=[[266.00,3.58,0],[0,0,1,0],[-1,0,-1,0],[9E9,9E9,9E9,9E9,9E9,9E9]];
    CONST robtarget p243:=[[261.47,-0.71,0],[0,0,1,0],[-1,0,-1,0],[9E9,9E9,9E9,9E9,9E9,9E9]];
    CONST robtarget p244:=[[260.16,-0.71,0],[0,0,1,0],[-1,0,-1,0],[9E9,9E9,9E9,9E9,9E9,9E9]];
    CONST robtarget p245:=[[256.20,-0.71,0],[0,0,1,0],[-1,0,-1,0],[9E9,9E9,9E9,9E9,9E9,9E9]];
    CONST robtarget p246:=[[253.36,-0.49,0],[0,0,1,0],[-1,0,-1,0],[9E9,9E9,9E9,9E9,9E9,9E9]];
    CONST robtarget p247:=[[249.24,0.15,0],[0,0,1,0],[-1,0,-1,0],[9E9,9E9,9E9,9E9,9E9,9E9]];
    CONST robtarget p248:=[[248.58,0.36,0],[0,0,1,0],[-1,0,-1,0],[9E9,9E9,9E9,9E9,9E9,9E9]];
    CONST robtarget p249:=[[246.61,1.00,0],[0,0,1,0],[-1,0,-1,0],[9E9,9E9,9E9,9E9,9E9,9E9]];
    CONST robtarget p250:=[[246.61,5.64,0],[0,0,1,0],[-1,0,-1,0],[9E9,9E9,9E9,9E9,9E9,9E9]];
    CONST robtarget p251:=[[249.68,4.35,0],[0,0,1,0],[-1,0,-1,0],[9E9,9E9,9E9,9E9,9E9,9E9]];
    CONST robtarget p252:=[[253.93,3.05,0],[0,0,1,0],[-1,0,-1,0],[9E9,9E9,9E9,9E9,9E9,9E9]];
    CONST robtarget p253:=[[254.52,3.05,0],[0,0,1,0],[-1,0,-1,0],[9E9,9E9,9E9,9E9,9E9,9E9]];
    CONST robtarget p254:=[[256.30,3.05,0],[0,0,1,0],[-1,0,-1,0],[9E9,9E9,9E9,9E9,9E9,9E9]];
    CONST robtarget p255:=[[259.53,3.59,0],[0,0,1,0],[-1,0,-1,0],[9E9,9E9,9E9,9E9,9E9,9E9]];
    CONST robtarget p256:=[[262.89,5.22,0],[0,0,1,0],[-1,0,-1,0],[9E9,9E9,9E9,9E9,9E9,9E9]];
    CONST robtarget p257:=[[262.89,5.72,0],[0,0,1,0],[-1,0,-1,0],[9E9,9E9,9E9,9E9,9E9,9E9]];
    CONST robtarget p258:=[[262.89,7.20,0],[0,0,1,0],[-1,0,-1,0],[9E9,9E9,9E9,9E9,9E9,9E9]];
    CONST robtarget p259:=[[262.27,9.06,0],[0,0,1,0],[-1,0,-1,0],[9E9,9E9,9E9,9E9,9E9,9E9]];
    CONST robtarget p260:=[[260.42,10.99,0],[0,0,1,0],[-1,0,-1,0],[9E9,9E9,9E9,9E9,9E9,9E9]];
    CONST robtarget p261:=[[259.38,11.21,0],[0,0,1,0],[-1,0,-1,0],[9E9,9E9,9E9,9E9,9E9,9E9]];
    CONST robtarget p262:=[[256.25,11.89,0],[0,0,1,0],[-1,0,-1,0],[9E9,9E9,9E9,9E9,9E9,9E9]];
    CONST robtarget p263:=[[254.69,12.26,0],[0,0,1,0],[-1,0,-1,0],[9E9,9E9,9E9,9E9,9E9,9E9]];
    CONST robtarget p264:=[[250.63,13.82,0],[0,0,1,0],[-1,0,-1,0],[9E9,9E9,9E9,9E9,9E9,9E9]];
    CONST robtarget p265:=[[246.80,16.77,0],[0,0,1,0],[-1,0,-1,0],[9E9,9E9,9E9,9E9,9E9,9E9]];
    CONST robtarget p266:=[[246.80,17.57,0],[0,0,1,0],[-1,0,-1,0],[9E9,9E9,9E9,9E9,9E9,9E9]];
    CONST robtarget p267:=[[246.80,19.95,0],[0,0,1,0],[-1,0,-1,0],[9E9,9E9,9E9,9E9,9E9,9E9]];
    CONST robtarget p268:=[[248.17,23.89,0],[0,0,1,0],[-1,0,-1,0],[9E9,9E9,9E9,9E9,9E9,9E9]];
    CONST robtarget p269:=[[252.27,28.00,0],[0,0,1,0],[-1,0,-1,0],[9E9,9E9,9E9,9E9,9E9,9E9]];
    CONST robtarget p270:=[[253.53,28.00,0],[0,0,1,0],[-1,0,-1,0],[9E9,9E9,9E9,9E9,9E9,9E9]];
    CONST robtarget p271:=[[257.30,28.00,0],[0,0,1,0],[-1,0,-1,0],[9E9,9E9,9E9,9E9,9E9,9E9]];
    CONST robtarget p272:=[[260.27,27.82,0],[0,0,1,0],[-1,0,-1,0],[9E9,9E9,9E9,9E9,9E9,9E9]];
    CONST robtarget p273:=[[264.18,27.27,0],[0,0,1,0],[-1,0,-1,0],[9E9,9E9,9E9,9E9,9E9,9E9]];
    CONST robtarget p274:=[[264.65,27.09,0],[0,0,1,0],[-1,0,-1,0],[9E9,9E9,9E9,9E9,9E9,9E9]];
    CONST robtarget p275:=[[266.04,26.54,0],[0,0,1,0],[-1,0,-1,0],[9E9,9E9,9E9,9E9,9E9,9E9]];
    ! Path 16/26
    CONST robtarget p276:=[[279.10,35.11,0],[0,0,1,0],[-1,0,-1,0],[9E9,9E9,9E9,9E9,9E9,9E9]];
    CONST robtarget p277:=[[279.10,27.34,0],[0,0,1,0],[-1,0,-1,0],[9E9,9E9,9E9,9E9,9E9,9E9]];
    CONST robtarget p278:=[[288.35,27.34,0],[0,0,1,0],[-1,0,-1,0],[9E9,9E9,9E9,9E9,9E9,9E9]];
    CONST robtarget p279:=[[288.35,23.85,0],[0,0,1,0],[-1,0,-1,0],[9E9,9E9,9E9,9E9,9E9,9E9]];
    CONST robtarget p280:=[[279.10,23.85,0],[0,0,1,0],[-1,0,-1,0],[9E9,9E9,9E9,9E9,9E9,9E9]];
    CONST robtarget p281:=[[279.10,9.01,0],[0,0,1,0],[-1,0,-1,0],[9E9,9E9,9E9,9E9,9E9,9E9]];
    CONST robtarget p282:=[[279.56,6.02,0],[0,0,1,0],[-1,0,-1,0],[9E9,9E9,9E9,9E9,9E9,9E9]];
    CONST robtarget p283:=[[280.93,3.76,0],[0,0,1,0],[-1,0,-1,0],[9E9,9E9,9E9,9E9,9E9,9E9]];
    CONST robtarget p284:=[[281.63,3.76,0],[0,0,1,0],[-1,0,-1,0],[9E9,9E9,9E9,9E9,9E9,9E9]];
    CONST robtarget p285:=[[283.74,3.76,0],[0,0,1,0],[-1,0,-1,0],[9E9,9E9,9E9,9E9,9E9,9E9]];
    CONST robtarget p286:=[[288.35,3.76,0],[0,0,1,0],[-1,0,-1,0],[9E9,9E9,9E9,9E9,9E9,9E9]];
    CONST robtarget p287:=[[288.35,0.00,0],[0,0,1,0],[-1,0,-1,0],[9E9,9E9,9E9,9E9,9E9,9E9]];
    CONST robtarget p288:=[[283.74,0.00,0],[0,0,1,0],[-1,0,-1,0],[9E9,9E9,9E9,9E9,9E9,9E9]];
    CONST robtarget p289:=[[278.85,0.97,0],[0,0,1,0],[-1,0,-1,0],[9E9,9E9,9E9,9E9,9E9,9E9]];
    CONST robtarget p290:=[[274.58,3.88,0],[0,0,1,0],[-1,0,-1,0],[9E9,9E9,9E9,9E9,9E9,9E9]];
    CONST robtarget p291:=[[274.58,5.16,0],[0,0,1,0],[-1,0,-1,0],[9E9,9E9,9E9,9E9,9E9,9E9]];
    CONST robtarget p292:=[[274.58,9.01,0],[0,0,1,0],[-1,0,-1,0],[9E9,9E9,9E9,9E9,9E9,9E9]];
    CONST robtarget p293:=[[274.58,23.85,0],[0,0,1,0],[-1,0,-1,0],[9E9,9E9,9E9,9E9,9E9,9E9]];
    CONST robtarget p294:=[[271.29,23.85,0],[0,0,1,0],[-1,0,-1,0],[9E9,9E9,9E9,9E9,9E9,9E9]];
    CONST robtarget p295:=[[271.29,27.34,0],[0,0,1,0],[-1,0,-1,0],[9E9,9E9,9E9,9E9,9E9,9E9]];
    CONST robtarget p296:=[[274.58,27.34,0],[0,0,1,0],[-1,0,-1,0],[9E9,9E9,9E9,9E9,9E9,9E9]];
    CONST robtarget p297:=[[274.58,35.11,0],[0,0,1,0],[-1,0,-1,0],[9E9,9E9,9E9,9E9,9E9,9E9]];
    CONST robtarget p298:=[[279.10,35.11,0],[0,0,1,0],[-1,0,-1,0],[9E9,9E9,9E9,9E9,9E9,9E9]];
    ! Path 17/26
    CONST robtarget p299:=[[317.65,14.79,0],[0,0,1,0],[-1,0,-1,0],[9E9,9E9,9E9,9E9,9E9,9E9]];
    CONST robtarget p300:=[[317.65,12.60,0],[0,0,1,0],[-1,0,-1,0],[9E9,9E9,9E9,9E9,9E9,9E9]];
    CONST robtarget p301:=[[297.00,12.60,0],[0,0,1,0],[-1,0,-1,0],[9E9,9E9,9E9,9E9,9E9,9E9]];
    CONST robtarget p302:=[[298.47,7.90,0],[0,0,1,0],[-1,0,-1,0],[9E9,9E9,9E9,9E9,9E9,9E9]];
    CONST robtarget p303:=[[302.29,3.10,0],[0,0,1,0],[-1,0,-1,0],[9E9,9E9,9E9,9E9,9E9,9E9]];
    CONST robtarget p304:=[[303.41,3.10,0],[0,0,1,0],[-1,0,-1,0],[9E9,9E9,9E9,9E9,9E9,9E9]];
    CONST robtarget p305:=[[306.76,3.10,0],[0,0,1,0],[-1,0,-1,0],[9E9,9E9,9E9,9E9,9E9,9E9]];
    CONST robtarget p306:=[[309.92,3.42,0],[0,0,1,0],[-1,0,-1,0],[9E9,9E9,9E9,9E9,9E9,9E9]];
    CONST robtarget p307:=[[314.21,4.37,0],[0,0,1,0],[-1,0,-1,0],[9E9,9E9,9E9,9E9,9E9,9E9]];
    CONST robtarget p308:=[[314.81,4.69,0],[0,0,1,0],[-1,0,-1,0],[9E9,9E9,9E9,9E9,9E9,9E9]];
    CONST robtarget p309:=[[316.60,5.64,0],[0,0,1,0],[-1,0,-1,0],[9E9,9E9,9E9,9E9,9E9,9E9]];
    CONST robtarget p310:=[[316.60,1.39,0],[0,0,1,0],[-1,0,-1,0],[9E9,9E9,9E9,9E9,9E9,9E9]];
    CONST robtarget p311:=[[313.52,0.35,0],[0,0,1,0],[-1,0,-1,0],[9E9,9E9,9E9,9E9,9E9,9E9]];
    CONST robtarget p312:=[[309.11,-0.71,0],[0,0,1,0],[-1,0,-1,0],[9E9,9E9,9E9,9E9,9E9,9E9]];
    CONST robtarget p313:=[[308.45,-0.71,0],[0,0,1,0],[-1,0,-1,0],[9E9,9E9,9E9,9E9,9E9,9E9]];
    CONST robtarget p314:=[[306.49,-0.71,0],[0,0,1,0],[-1,0,-1,0],[9E9,9E9,9E9,9E9,9E9,9E9]];
    CONST robtarget p315:=[[302.01,0.14,0],[0,0,1,0],[-1,0,-1,0],[9E9,9E9,9E9,9E9,9E9,9E9]];
    CONST robtarget p316:=[[297.28,2.68,0],[0,0,1,0],[-1,0,-1,0],[9E9,9E9,9E9,9E9,9E9,9E9]];
    CONST robtarget p317:=[[292.31,6.91,0],[0,0,1,0],[-1,0,-1,0],[9E9,9E9,9E9,9E9,9E9,9E9]];
    CONST robtarget p318:=[[292.31,8.53,0],[0,0,1,0],[-1,0,-1,0],[9E9,9E9,9E9,9E9,9E9,9E9]];
    CONST robtarget p319:=[[292.31,13.40,0],[0,0,1,0],[-1,0,-1,0],[9E9,9E9,9E9,9E9,9E9,9E9]];
    CONST robtarget p320:=[[293.12,18.01,0],[0,0,1,0],[-1,0,-1,0],[9E9,9E9,9E9,9E9,9E9,9E9]];
    CONST robtarget p321:=[[295.53,22.88,0],[0,0,1,0],[-1,0,-1,0],[9E9,9E9,9E9,9E9,9E9,9E9]];
    CONST robtarget p322:=[[299.56,28.00,0],[0,0,1,0],[-1,0,-1,0],[9E9,9E9,9E9,9E9,9E9,9E9]];
    CONST robtarget p323:=[[301.10,28.00,0],[0,0,1,0],[-1,0,-1,0],[9E9,9E9,9E9,9E9,9E9,9E9]];
    CONST robtarget p324:=[[305.71,28.00,0],[0,0,1,0],[-1,0,-1,0],[9E9,9E9,9E9,9E9,9E9,9E9]];
    CONST robtarget p325:=[[309.49,27.21,0],[0,0,1,0],[-1,0,-1,0],[9E9,9E9,9E9,9E9,9E9,9E9]];
    CONST robtarget p326:=[[313.47,24.85,0],[0,0,1,0],[-1,0,-1,0],[9E9,9E9,9E9,9E9,9E9,9E9]];
    CONST robtarget p327:=[[317.65,20.90,0],[0,0,1,0],[-1,0,-1,0],[9E9,9E9,9E9,9E9,9E9,9E9]];
    CONST robtarget p328:=[[317.65,19.37,0],[0,0,1,0],[-1,0,-1,0],[9E9,9E9,9E9,9E9,9E9,9E9]];
    CONST robtarget p329:=[[317.65,14.79,0],[0,0,1,0],[-1,0,-1,0],[9E9,9E9,9E9,9E9,9E9,9E9]];
    ! Path 18/26
    CONST robtarget p330:=[[313.16,16.11,0],[0,0,1,0],[-1,0,-1,0],[9E9,9E9,9E9,9E9,9E9,9E9]];
    CONST robtarget p331:=[[312.12,19.98,0],[0,0,1,0],[-1,0,-1,0],[9E9,9E9,9E9,9E9,9E9,9E9]];
    CONST robtarget p332:=[[309.08,24.19,0],[0,0,1,0],[-1,0,-1,0],[9E9,9E9,9E9,9E9,9E9,9E9]];
    CONST robtarget p333:=[[308.25,24.19,0],[0,0,1,0],[-1,0,-1,0],[9E9,9E9,9E9,9E9,9E9,9E9]];
    CONST robtarget p334:=[[305.76,24.19,0],[0,0,1,0],[-1,0,-1,0],[9E9,9E9,9E9,9E9,9E9,9E9]];
    CONST robtarget p335:=[[301.81,23.13,0],[0,0,1,0],[-1,0,-1,0],[9E9,9E9,9E9,9E9,9E9,9E9]];
    CONST robtarget p336:=[[297.49,19.95,0],[0,0,1,0],[-1,0,-1,0],[9E9,9E9,9E9,9E9,9E9,9E9]];
    CONST robtarget p337:=[[297.40,18.98,0],[0,0,1,0],[-1,0,-1,0],[9E9,9E9,9E9,9E9,9E9,9E9]];
    CONST robtarget p338:=[[297.14,16.09,0],[0,0,1,0],[-1,0,-1,0],[9E9,9E9,9E9,9E9,9E9,9E9]];
    CONST robtarget p339:=[[313.16,16.11,0],[0,0,1,0],[-1,0,-1,0],[9E9,9E9,9E9,9E9,9E9,9E9]];
    ! Path 19/26
    CONST robtarget p340:=[[340.87,23.14,0],[0,0,1,0],[-1,0,-1,0],[9E9,9E9,9E9,9E9,9E9,9E9]];
    CONST robtarget p341:=[[339.86,23.58,0],[0,0,1,0],[-1,0,-1,0],[9E9,9E9,9E9,9E9,9E9,9E9]];
    CONST robtarget p342:=[[338.33,24.00,0],[0,0,1,0],[-1,0,-1,0],[9E9,9E9,9E9,9E9,9E9,9E9]];
    CONST robtarget p343:=[[338.06,24.00,0],[0,0,1,0],[-1,0,-1,0],[9E9,9E9,9E9,9E9,9E9,9E9]];
    CONST robtarget p344:=[[337.26,24.00,0],[0,0,1,0],[-1,0,-1,0],[9E9,9E9,9E9,9E9,9E9,9E9]];
    CONST robtarget p345:=[[333.38,22.76,0],[0,0,1,0],[-1,0,-1,0],[9E9,9E9,9E9,9E9,9E9,9E9]];
    CONST robtarget p346:=[[329.37,19.04,0],[0,0,1,0],[-1,0,-1,0],[9E9,9E9,9E9,9E9,9E9,9E9]];
    CONST robtarget p347:=[[329.37,17.88,0],[0,0,1,0],[-1,0,-1,0],[9E9,9E9,9E9,9E9,9E9,9E9]];
    CONST robtarget p348:=[[329.37,14.40,0],[0,0,1,0],[-1,0,-1,0],[9E9,9E9,9E9,9E9,9E9,9E9]];
    CONST robtarget p349:=[[329.37,0.00,0],[0,0,1,0],[-1,0,-1,0],[9E9,9E9,9E9,9E9,9E9,9E9]];
    CONST robtarget p350:=[[324.85,0.00,0],[0,0,1,0],[-1,0,-1,0],[9E9,9E9,9E9,9E9,9E9,9E9]];
    CONST robtarget p351:=[[324.85,27.34,0],[0,0,1,0],[-1,0,-1,0],[9E9,9E9,9E9,9E9,9E9,9E9]];
    CONST robtarget p352:=[[329.37,27.34,0],[0,0,1,0],[-1,0,-1,0],[9E9,9E9,9E9,9E9,9E9,9E9]];
    CONST robtarget p353:=[[329.37,23.10,0],[0,0,1,0],[-1,0,-1,0],[9E9,9E9,9E9,9E9,9E9,9E9]];
    CONST robtarget p354:=[[331.57,25.57,0],[0,0,1,0],[-1,0,-1,0],[9E9,9E9,9E9,9E9,9E9,9E9]];
    CONST robtarget p355:=[[335.33,28.00,0],[0,0,1,0],[-1,0,-1,0],[9E9,9E9,9E9,9E9,9E9,9E9]];
    CONST robtarget p356:=[[336.14,28.00,0],[0,0,1,0],[-1,0,-1,0],[9E9,9E9,9E9,9E9,9E9,9E9]];
    CONST robtarget p357:=[[338.57,28.00,0],[0,0,1,0],[-1,0,-1,0],[9E9,9E9,9E9,9E9,9E9,9E9]];
    CONST robtarget p358:=[[339.20,27.97,0],[0,0,1,0],[-1,0,-1,0],[9E9,9E9,9E9,9E9,9E9,9E9]];
    CONST robtarget p359:=[[340.16,27.88,0],[0,0,1,0],[-1,0,-1,0],[9E9,9E9,9E9,9E9,9E9,9E9]];
    CONST robtarget p360:=[[340.33,27.85,0],[0,0,1,0],[-1,0,-1,0],[9E9,9E9,9E9,9E9,9E9,9E9]];
    CONST robtarget p361:=[[340.84,27.76,0],[0,0,1,0],[-1,0,-1,0],[9E9,9E9,9E9,9E9,9E9,9E9]];
    CONST robtarget p362:=[[340.87,23.14,0],[0,0,1,0],[-1,0,-1,0],[9E9,9E9,9E9,9E9,9E9,9E9]];
    ! Path 20/26
    CONST robtarget p363:=[[366.36,4.15,0],[0,0,1,0],[-1,0,-1,0],[9E9,9E9,9E9,9E9,9E9,9E9]];
    CONST robtarget p364:=[[383.57,4.15,0],[0,0,1,0],[-1,0,-1,0],[9E9,9E9,9E9,9E9,9E9,9E9]];
    CONST robtarget p365:=[[383.57,0.00,0],[0,0,1,0],[-1,0,-1,0],[9E9,9E9,9E9,9E9,9E9,9E9]];
    CONST robtarget p366:=[[360.42,0.00,0],[0,0,1,0],[-1,0,-1,0],[9E9,9E9,9E9,9E9,9E9,9E9]];
    CONST robtarget p367:=[[360.42,4.15,0],[0,0,1,0],[-1,0,-1,0],[9E9,9E9,9E9,9E9,9E9,9E9]];
    CONST robtarget p368:=[[363.06,6.85,0],[0,0,1,0],[-1,0,-1,0],[9E9,9E9,9E9,9E9,9E9,9E9]];
    CONST robtarget p369:=[[367.23,11.08,0],[0,0,1,0],[-1,0,-1,0],[9E9,9E9,9E9,9E9,9E9,9E9]];
    CONST robtarget p370:=[[372.92,16.85,0],[0,0,1,0],[-1,0,-1,0],[9E9,9E9,9E9,9E9,9E9,9E9]];
    CONST robtarget p371:=[[373.24,17.20,0],[0,0,1,0],[-1,0,-1,0],[9E9,9E9,9E9,9E9,9E9,9E9]];
    CONST robtarget p372:=[[374.17,18.26,0],[0,0,1,0],[-1,0,-1,0],[9E9,9E9,9E9,9E9,9E9,9E9]];
    CONST robtarget p373:=[[376.42,21.18,0],[0,0,1,0],[-1,0,-1,0],[9E9,9E9,9E9,9E9,9E9,9E9]];
    CONST robtarget p374:=[[378.42,24.61,0],[0,0,1,0],[-1,0,-1,0],[9E9,9E9,9E9,9E9,9E9,9E9]];
    CONST robtarget p375:=[[378.42,25.05,0],[0,0,1,0],[-1,0,-1,0],[9E9,9E9,9E9,9E9,9E9,9E9]];
    CONST robtarget p376:=[[378.42,26.39,0],[0,0,1,0],[-1,0,-1,0],[9E9,9E9,9E9,9E9,9E9,9E9]];
    CONST robtarget p377:=[[377.40,29.49,0],[0,0,1,0],[-1,0,-1,0],[9E9,9E9,9E9,9E9,9E9,9E9]];
    CONST robtarget p378:=[[374.34,32.96,0],[0,0,1,0],[-1,0,-1,0],[9E9,9E9,9E9,9E9,9E9,9E9]];
    CONST robtarget p379:=[[373.52,32.96,0],[0,0,1,0],[-1,0,-1,0],[9E9,9E9,9E9,9E9,9E9,9E9]];
    CONST robtarget p380:=[[371.07,32.96,0],[0,0,1,0],[-1,0,-1,0],[9E9,9E9,9E9,9E9,9E9,9E9]];
    CONST robtarget p381:=[[368.04,32.56,0],[0,0,1,0],[-1,0,-1,0],[9E9,9E9,9E9,9E9,9E9,9E9]];
    CONST robtarget p382:=[[363.60,31.35,0],[0,0,1,0],[-1,0,-1,0],[9E9,9E9,9E9,9E9,9E9,9E9]];
    CONST robtarget p383:=[[362.87,30.94,0],[0,0,1,0],[-1,0,-1,0],[9E9,9E9,9E9,9E9,9E9,9E9]];
    CONST robtarget p384:=[[360.67,29.71,0],[0,0,1,0],[-1,0,-1,0],[9E9,9E9,9E9,9E9,9E9,9E9]];
    CONST robtarget p385:=[[360.67,34.69,0],[0,0,1,0],[-1,0,-1,0],[9E9,9E9,9E9,9E9,9E9,9E9]];
    CONST robtarget p386:=[[364.20,35.89,0],[0,0,1,0],[-1,0,-1,0],[9E9,9E9,9E9,9E9,9E9,9E9]];
    CONST robtarget p387:=[[368.82,37.11,0],[0,0,1,0],[-1,0,-1,0],[9E9,9E9,9E9,9E9,9E9,9E9]];
    CONST robtarget p388:=[[369.36,37.11,0],[0,0,1,0],[-1,0,-1,0],[9E9,9E9,9E9,9E9,9E9,9E9]];
    CONST robtarget p389:=[[370.97,37.11,0],[0,0,1,0],[-1,0,-1,0],[9E9,9E9,9E9,9E9,9E9,9E9]];
    CONST robtarget p390:=[[376.90,35.69,0],[0,0,1,0],[-1,0,-1,0],[9E9,9E9,9E9,9E9,9E9,9E9]];
    CONST robtarget p391:=[[383.37,31.45,0],[0,0,1,0],[-1,0,-1,0],[9E9,9E9,9E9,9E9,9E9,9E9]];
    CONST robtarget p392:=[[383.37,30.26,0],[0,0,1,0],[-1,0,-1,0],[9E9,9E9,9E9,9E9,9E9,9E9]];
    CONST robtarget p393:=[[383.37,26.71,0],[0,0,1,0],[-1,0,-1,0],[9E9,9E9,9E9,9E9,9E9,9E9]];
    CONST robtarget p394:=[[382.95,24.02,0],[0,0,1,0],[-1,0,-1,0],[9E9,9E9,9E9,9E9,9E9,9E9]];
    CONST robtarget p395:=[[381.69,20.43,0],[0,0,1,0],[-1,0,-1,0],[9E9,9E9,9E9,9E9,9E9,9E9]];
    CONST robtarget p396:=[[381.13,19.75,0],[0,0,1,0],[-1,0,-1,0],[9E9,9E9,9E9,9E9,9E9,9E9]];
    CONST robtarget p397:=[[379.47,17.70,0],[0,0,1,0],[-1,0,-1,0],[9E9,9E9,9E9,9E9,9E9,9E9]];
    CONST robtarget p398:=[[377.37,15.48,0],[0,0,1,0],[-1,0,-1,0],[9E9,9E9,9E9,9E9,9E9,9E9]];
    CONST robtarget p399:=[[372.31,10.23,0],[0,0,1,0],[-1,0,-1,0],[9E9,9E9,9E9,9E9,9E9,9E9]];
    CONST robtarget p400:=[[370.83,8.71,0],[0,0,1,0],[-1,0,-1,0],[9E9,9E9,9E9,9E9,9E9,9E9]];
    CONST robtarget p401:=[[366.36,4.15,0],[0,0,1,0],[-1,0,-1,0],[9E9,9E9,9E9,9E9,9E9,9E9]];
    ! Path 21/26
    CONST robtarget p402:=[[404.47,33.20,0],[0,0,1,0],[-1,0,-1,0],[9E9,9E9,9E9,9E9,9E9,9E9]];
    CONST robtarget p403:=[[400.65,31.33,0],[0,0,1,0],[-1,0,-1,0],[9E9,9E9,9E9,9E9,9E9,9E9]];
    CONST robtarget p404:=[[396.83,25.71,0],[0,0,1,0],[-1,0,-1,0],[9E9,9E9,9E9,9E9,9E9,9E9]];
    CONST robtarget p405:=[[396.83,23.83,0],[0,0,1,0],[-1,0,-1,0],[9E9,9E9,9E9,9E9,9E9,9E9]];
    CONST robtarget p406:=[[396.83,18.19,0],[0,0,1,0],[-1,0,-1,0],[9E9,9E9,9E9,9E9,9E9,9E9]];
    CONST robtarget p407:=[[397.25,13.19,0],[0,0,1,0],[-1,0,-1,0],[9E9,9E9,9E9,9E9,9E9,9E9]];
    CONST robtarget p408:=[[398.53,8.19,0],[0,0,1,0],[-1,0,-1,0],[9E9,9E9,9E9,9E9,9E9,9E9]];
    CONST robtarget p409:=[[400.66,3.20,0],[0,0,1,0],[-1,0,-1,0],[9E9,9E9,9E9,9E9,9E9,9E9]];
    CONST robtarget p410:=[[401.61,3.20,0],[0,0,1,0],[-1,0,-1,0],[9E9,9E9,9E9,9E9,9E9,9E9]];
    CONST robtarget p411:=[[404.47,3.20,0],[0,0,1,0],[-1,0,-1,0],[9E9,9E9,9E9,9E9,9E9,9E9]];
    CONST robtarget p412:=[[408.30,5.07,0],[0,0,1,0],[-1,0,-1,0],[9E9,9E9,9E9,9E9,9E9,9E9]];
    CONST robtarget p413:=[[412.13,10.69,0],[0,0,1,0],[-1,0,-1,0],[9E9,9E9,9E9,9E9,9E9,9E9]];
    CONST robtarget p414:=[[412.13,12.57,0],[0,0,1,0],[-1,0,-1,0],[9E9,9E9,9E9,9E9,9E9,9E9]];
    CONST robtarget p415:=[[412.13,18.19,0],[0,0,1,0],[-1,0,-1,0],[9E9,9E9,9E9,9E9,9E9,9E9]];
    CONST robtarget p416:=[[411.71,23.20,0],[0,0,1,0],[-1,0,-1,0],[9E9,9E9,9E9,9E9,9E9,9E9]];
    CONST robtarget p417:=[[410.43,28.20,0],[0,0,1,0],[-1,0,-1,0],[9E9,9E9,9E9,9E9,9E9,9E9]];
    CONST robtarget p418:=[[408.30,33.20,0],[0,0,1,0],[-1,0,-1,0],[9E9,9E9,9E9,9E9,9E9,9E9]];
    CONST robtarget p419:=[[407.34,33.20,0],[0,0,1,0],[-1,0,-1,0],[9E9,9E9,9E9,9E9,9E9,9E9]];
    CONST robtarget p420:=[[404.47,33.20,0],[0,0,1,0],[-1,0,-1,0],[9E9,9E9,9E9,9E9,9E9,9E9]];
    ! Path 22/26
    CONST robtarget p421:=[[404.47,37.11,0],[0,0,1,0],[-1,0,-1,0],[9E9,9E9,9E9,9E9,9E9,9E9]];
    CONST robtarget p422:=[[408.59,36.03,0],[0,0,1,0],[-1,0,-1,0],[9E9,9E9,9E9,9E9,9E9,9E9]];
    CONST robtarget p423:=[[412.79,32.80,0],[0,0,1,0],[-1,0,-1,0],[9E9,9E9,9E9,9E9,9E9,9E9]];
    CONST robtarget p424:=[[417.07,27.42,0],[0,0,1,0],[-1,0,-1,0],[9E9,9E9,9E9,9E9,9E9,9E9]];
    CONST robtarget p425:=[[417.07,25.11,0],[0,0,1,0],[-1,0,-1,0],[9E9,9E9,9E9,9E9,9E9,9E9]];
    CONST robtarget p426:=[[417.07,18.19,0],[0,0,1,0],[-1,0,-1,0],[9E9,9E9,9E9,9E9,9E9,9E9]];
    CONST robtarget p427:=[[416.66,13.56,0],[0,0,1,0],[-1,0,-1,0],[9E9,9E9,9E9,9E9,9E9,9E9]];
    CONST robtarget p428:=[[415.45,8.86,0],[0,0,1,0],[-1,0,-1,0],[9E9,9E9,9E9,9E9,9E9,9E9]];
    CONST robtarget p429:=[[413.43,4.11,0],[0,0,1,0],[-1,0,-1,0],[9E9,9E9,9E9,9E9,9E9,9E9]];
    CONST robtarget p430:=[[410.60,-0.71,0],[0,0,1,0],[-1,0,-1,0],[9E9,9E9,9E9,9E9,9E9,9E9]];
    CONST robtarget p431:=[[409.06,-0.71,0],[0,0,1,0],[-1,0,-1,0],[9E9,9E9,9E9,9E9,9E9,9E9]];
    CONST robtarget p432:=[[404.47,-0.71,0],[0,0,1,0],[-1,0,-1,0],[9E9,9E9,9E9,9E9,9E9,9E9]];
    CONST robtarget p433:=[[400.34,0.37,0],[0,0,1,0],[-1,0,-1,0],[9E9,9E9,9E9,9E9,9E9,9E9]];
    CONST robtarget p434:=[[396.15,3.60,0],[0,0,1,0],[-1,0,-1,0],[9E9,9E9,9E9,9E9,9E9,9E9]];
    CONST robtarget p435:=[[391.87,8.98,0],[0,0,1,0],[-1,0,-1,0],[9E9,9E9,9E9,9E9,9E9,9E9]];
    CONST robtarget p436:=[[391.87,11.29,0],[0,0,1,0],[-1,0,-1,0],[9E9,9E9,9E9,9E9,9E9,9E9]];
    CONST robtarget p437:=[[391.87,18.19,0],[0,0,1,0],[-1,0,-1,0],[9E9,9E9,9E9,9E9,9E9,9E9]];
    CONST robtarget p438:=[[392.27,22.83,0],[0,0,1,0],[-1,0,-1,0],[9E9,9E9,9E9,9E9,9E9,9E9]];
    CONST robtarget p439:=[[393.49,27.53,0],[0,0,1,0],[-1,0,-1,0],[9E9,9E9,9E9,9E9,9E9,9E9]];
    CONST robtarget p440:=[[395.51,32.29,0],[0,0,1,0],[-1,0,-1,0],[9E9,9E9,9E9,9E9,9E9,9E9]];
    CONST robtarget p441:=[[398.34,37.11,0],[0,0,1,0],[-1,0,-1,0],[9E9,9E9,9E9,9E9,9E9,9E9]];
    CONST robtarget p442:=[[399.87,37.11,0],[0,0,1,0],[-1,0,-1,0],[9E9,9E9,9E9,9E9,9E9,9E9]];
    CONST robtarget p443:=[[404.47,37.11,0],[0,0,1,0],[-1,0,-1,0],[9E9,9E9,9E9,9E9,9E9,9E9]];
    ! Path 23/26
    CONST robtarget p444:=[[436.28,33.20,0],[0,0,1,0],[-1,0,-1,0],[9E9,9E9,9E9,9E9,9E9,9E9]];
    CONST robtarget p445:=[[432.46,31.33,0],[0,0,1,0],[-1,0,-1,0],[9E9,9E9,9E9,9E9,9E9,9E9]];
    CONST robtarget p446:=[[428.64,25.71,0],[0,0,1,0],[-1,0,-1,0],[9E9,9E9,9E9,9E9,9E9,9E9]];
    CONST robtarget p447:=[[428.64,23.83,0],[0,0,1,0],[-1,0,-1,0],[9E9,9E9,9E9,9E9,9E9,9E9]];
    CONST robtarget p448:=[[428.64,18.19,0],[0,0,1,0],[-1,0,-1,0],[9E9,9E9,9E9,9E9,9E9,9E9]];
    CONST robtarget p449:=[[429.06,13.19,0],[0,0,1,0],[-1,0,-1,0],[9E9,9E9,9E9,9E9,9E9,9E9]];
    CONST robtarget p450:=[[430.34,8.19,0],[0,0,1,0],[-1,0,-1,0],[9E9,9E9,9E9,9E9,9E9,9E9]];
    CONST robtarget p451:=[[432.47,3.20,0],[0,0,1,0],[-1,0,-1,0],[9E9,9E9,9E9,9E9,9E9,9E9]];
    CONST robtarget p452:=[[433.42,3.20,0],[0,0,1,0],[-1,0,-1,0],[9E9,9E9,9E9,9E9,9E9,9E9]];
    CONST robtarget p453:=[[436.28,3.20,0],[0,0,1,0],[-1,0,-1,0],[9E9,9E9,9E9,9E9,9E9,9E9]];
    CONST robtarget p454:=[[440.11,5.07,0],[0,0,1,0],[-1,0,-1,0],[9E9,9E9,9E9,9E9,9E9,9E9]];
    CONST robtarget p455:=[[443.95,10.69,0],[0,0,1,0],[-1,0,-1,0],[9E9,9E9,9E9,9E9,9E9,9E9]];
    CONST robtarget p456:=[[443.95,12.57,0],[0,0,1,0],[-1,0,-1,0],[9E9,9E9,9E9,9E9,9E9,9E9]];
    CONST robtarget p457:=[[443.95,18.19,0],[0,0,1,0],[-1,0,-1,0],[9E9,9E9,9E9,9E9,9E9,9E9]];
    CONST robtarget p458:=[[443.52,23.20,0],[0,0,1,0],[-1,0,-1,0],[9E9,9E9,9E9,9E9,9E9,9E9]];
    CONST robtarget p459:=[[442.24,28.20,0],[0,0,1,0],[-1,0,-1,0],[9E9,9E9,9E9,9E9,9E9,9E9]];
    CONST robtarget p460:=[[440.11,33.20,0],[0,0,1,0],[-1,0,-1,0],[9E9,9E9,9E9,9E9,9E9,9E9]];
    CONST robtarget p461:=[[439.15,33.20,0],[0,0,1,0],[-1,0,-1,0],[9E9,9E9,9E9,9E9,9E9,9E9]];
    CONST robtarget p462:=[[436.28,33.20,0],[0,0,1,0],[-1,0,-1,0],[9E9,9E9,9E9,9E9,9E9,9E9]];
    ! Path 24/26
    CONST robtarget p463:=[[436.28,37.11,0],[0,0,1,0],[-1,0,-1,0],[9E9,9E9,9E9,9E9,9E9,9E9]];
    CONST robtarget p464:=[[440.40,36.03,0],[0,0,1,0],[-1,0,-1,0],[9E9,9E9,9E9,9E9,9E9,9E9]];
    CONST robtarget p465:=[[444.60,32.80,0],[0,0,1,0],[-1,0,-1,0],[9E9,9E9,9E9,9E9,9E9,9E9]];
    CONST robtarget p466:=[[448.88,27.42,0],[0,0,1,0],[-1,0,-1,0],[9E9,9E9,9E9,9E9,9E9,9E9]];
    CONST robtarget p467:=[[448.88,25.11,0],[0,0,1,0],[-1,0,-1,0],[9E9,9E9,9E9,9E9,9E9,9E9]];
    CONST robtarget p468:=[[448.88,18.19,0],[0,0,1,0],[-1,0,-1,0],[9E9,9E9,9E9,9E9,9E9,9E9]];
    CONST robtarget p469:=[[448.47,13.56,0],[0,0,1,0],[-1,0,-1,0],[9E9,9E9,9E9,9E9,9E9,9E9]];
    CONST robtarget p470:=[[447.26,8.86,0],[0,0,1,0],[-1,0,-1,0],[9E9,9E9,9E9,9E9,9E9,9E9]];
    CONST robtarget p471:=[[445.24,4.11,0],[0,0,1,0],[-1,0,-1,0],[9E9,9E9,9E9,9E9,9E9,9E9]];
    CONST robtarget p472:=[[442.41,-0.71,0],[0,0,1,0],[-1,0,-1,0],[9E9,9E9,9E9,9E9,9E9,9E9]];
    CONST robtarget p473:=[[440.88,-0.71,0],[0,0,1,0],[-1,0,-1,0],[9E9,9E9,9E9,9E9,9E9,9E9]];
    CONST robtarget p474:=[[436.28,-0.71,0],[0,0,1,0],[-1,0,-1,0],[9E9,9E9,9E9,9E9,9E9,9E9]];
    CONST robtarget p475:=[[432.16,0.37,0],[0,0,1,0],[-1,0,-1,0],[9E9,9E9,9E9,9E9,9E9,9E9]];
    CONST robtarget p476:=[[427.96,3.60,0],[0,0,1,0],[-1,0,-1,0],[9E9,9E9,9E9,9E9,9E9,9E9]];
    CONST robtarget p477:=[[423.68,8.98,0],[0,0,1,0],[-1,0,-1,0],[9E9,9E9,9E9,9E9,9E9,9E9]];
    CONST robtarget p478:=[[423.68,11.29,0],[0,0,1,0],[-1,0,-1,0],[9E9,9E9,9E9,9E9,9E9,9E9]];
    CONST robtarget p479:=[[423.68,18.19,0],[0,0,1,0],[-1,0,-1,0],[9E9,9E9,9E9,9E9,9E9,9E9]];
    CONST robtarget p480:=[[424.09,22.83,0],[0,0,1,0],[-1,0,-1,0],[9E9,9E9,9E9,9E9,9E9,9E9]];
    CONST robtarget p481:=[[425.30,27.53,0],[0,0,1,0],[-1,0,-1,0],[9E9,9E9,9E9,9E9,9E9,9E9]];
    CONST robtarget p482:=[[427.32,32.29,0],[0,0,1,0],[-1,0,-1,0],[9E9,9E9,9E9,9E9,9E9,9E9]];
    CONST robtarget p483:=[[430.15,37.11,0],[0,0,1,0],[-1,0,-1,0],[9E9,9E9,9E9,9E9,9E9,9E9]];
    CONST robtarget p484:=[[431.68,37.11,0],[0,0,1,0],[-1,0,-1,0],[9E9,9E9,9E9,9E9,9E9,9E9]];
    CONST robtarget p485:=[[436.28,37.11,0],[0,0,1,0],[-1,0,-1,0],[9E9,9E9,9E9,9E9,9E9,9E9]];
    ! Path 25/26
    CONST robtarget p486:=[[468.09,33.20,0],[0,0,1,0],[-1,0,-1,0],[9E9,9E9,9E9,9E9,9E9,9E9]];
    CONST robtarget p487:=[[464.28,31.33,0],[0,0,1,0],[-1,0,-1,0],[9E9,9E9,9E9,9E9,9E9,9E9]];
    CONST robtarget p488:=[[460.45,25.71,0],[0,0,1,0],[-1,0,-1,0],[9E9,9E9,9E9,9E9,9E9,9E9]];
    CONST robtarget p489:=[[460.45,23.83,0],[0,0,1,0],[-1,0,-1,0],[9E9,9E9,9E9,9E9,9E9,9E9]];
    CONST robtarget p490:=[[460.45,18.19,0],[0,0,1,0],[-1,0,-1,0],[9E9,9E9,9E9,9E9,9E9,9E9]];
    CONST robtarget p491:=[[460.88,13.19,0],[0,0,1,0],[-1,0,-1,0],[9E9,9E9,9E9,9E9,9E9,9E9]];
    CONST robtarget p492:=[[462.15,8.19,0],[0,0,1,0],[-1,0,-1,0],[9E9,9E9,9E9,9E9,9E9,9E9]];
    CONST robtarget p493:=[[464.28,3.20,0],[0,0,1,0],[-1,0,-1,0],[9E9,9E9,9E9,9E9,9E9,9E9]];
    CONST robtarget p494:=[[465.23,3.20,0],[0,0,1,0],[-1,0,-1,0],[9E9,9E9,9E9,9E9,9E9,9E9]];
    CONST robtarget p495:=[[468.09,3.20,0],[0,0,1,0],[-1,0,-1,0],[9E9,9E9,9E9,9E9,9E9,9E9]];
    CONST robtarget p496:=[[471.92,5.07,0],[0,0,1,0],[-1,0,-1,0],[9E9,9E9,9E9,9E9,9E9,9E9]];
    CONST robtarget p497:=[[475.76,10.69,0],[0,0,1,0],[-1,0,-1,0],[9E9,9E9,9E9,9E9,9E9,9E9]];
    CONST robtarget p498:=[[475.76,12.57,0],[0,0,1,0],[-1,0,-1,0],[9E9,9E9,9E9,9E9,9E9,9E9]];
    CONST robtarget p499:=[[475.76,18.19,0],[0,0,1,0],[-1,0,-1,0],[9E9,9E9,9E9,9E9,9E9,9E9]];
    CONST robtarget p500:=[[475.33,23.20,0],[0,0,1,0],[-1,0,-1,0],[9E9,9E9,9E9,9E9,9E9,9E9]];
    CONST robtarget p501:=[[474.05,28.20,0],[0,0,1,0],[-1,0,-1,0],[9E9,9E9,9E9,9E9,9E9,9E9]];
    CONST robtarget p502:=[[471.92,33.20,0],[0,0,1,0],[-1,0,-1,0],[9E9,9E9,9E9,9E9,9E9,9E9]];
    CONST robtarget p503:=[[470.97,33.20,0],[0,0,1,0],[-1,0,-1,0],[9E9,9E9,9E9,9E9,9E9,9E9]];
    CONST robtarget p504:=[[468.09,33.20,0],[0,0,1,0],[-1,0,-1,0],[9E9,9E9,9E9,9E9,9E9,9E9]];
    ! Path 26/26
    CONST robtarget p505:=[[468.09,37.11,0],[0,0,1,0],[-1,0,-1,0],[9E9,9E9,9E9,9E9,9E9,9E9]];
    CONST robtarget p506:=[[472.21,36.03,0],[0,0,1,0],[-1,0,-1,0],[9E9,9E9,9E9,9E9,9E9,9E9]];
    CONST robtarget p507:=[[476.41,32.80,0],[0,0,1,0],[-1,0,-1,0],[9E9,9E9,9E9,9E9,9E9,9E9]];
    CONST robtarget p508:=[[480.69,27.42,0],[0,0,1,0],[-1,0,-1,0],[9E9,9E9,9E9,9E9,9E9,9E9]];
    CONST robtarget p509:=[[480.69,25.11,0],[0,0,1,0],[-1,0,-1,0],[9E9,9E9,9E9,9E9,9E9,9E9]];
    CONST robtarget p510:=[[480.69,18.19,0],[0,0,1,0],[-1,0,-1,0],[9E9,9E9,9E9,9E9,9E9,9E9]];
    CONST robtarget p511:=[[480.28,13.56,0],[0,0,1,0],[-1,0,-1,0],[9E9,9E9,9E9,9E9,9E9,9E9]];
    CONST robtarget p512:=[[479.07,8.86,0],[0,0,1,0],[-1,0,-1,0],[9E9,9E9,9E9,9E9,9E9,9E9]];
    CONST robtarget p513:=[[477.05,4.11,0],[0,0,1,0],[-1,0,-1,0],[9E9,9E9,9E9,9E9,9E9,9E9]];
    CONST robtarget p514:=[[474.22,-0.71,0],[0,0,1,0],[-1,0,-1,0],[9E9,9E9,9E9,9E9,9E9,9E9]];
    CONST robtarget p515:=[[472.69,-0.71,0],[0,0,1,0],[-1,0,-1,0],[9E9,9E9,9E9,9E9,9E9,9E9]];
    CONST robtarget p516:=[[468.09,-0.71,0],[0,0,1,0],[-1,0,-1,0],[9E9,9E9,9E9,9E9,9E9,9E9]];
    CONST robtarget p517:=[[463.97,0.37,0],[0,0,1,0],[-1,0,-1,0],[9E9,9E9,9E9,9E9,9E9,9E9]];
    CONST robtarget p518:=[[459.77,3.60,0],[0,0,1,0],[-1,0,-1,0],[9E9,9E9,9E9,9E9,9E9,9E9]];
    CONST robtarget p519:=[[455.49,8.98,0],[0,0,1,0],[-1,0,-1,0],[9E9,9E9,9E9,9E9,9E9,9E9]];
    CONST robtarget p520:=[[455.49,11.29,0],[0,0,1,0],[-1,0,-1,0],[9E9,9E9,9E9,9E9,9E9,9E9]];
    CONST robtarget p521:=[[455.49,18.19,0],[0,0,1,0],[-1,0,-1,0],[9E9,9E9,9E9,9E9,9E9,9E9]];
    CONST robtarget p522:=[[455.90,22.83,0],[0,0,1,0],[-1,0,-1,0],[9E9,9E9,9E9,9E9,9E9,9E9]];
    CONST robtarget p523:=[[457.11,27.53,0],[0,0,1,0],[-1,0,-1,0],[9E9,9E9,9E9,9E9,9E9,9E9]];
    CONST robtarget p524:=[[459.13,32.29,0],[0,0,1,0],[-1,0,-1,0],[9E9,9E9,9E9,9E9,9E9,9E9]];
    CONST robtarget p525:=[[461.96,37.11,0],[0,0,1,0],[-1,0,-1,0],[9E9,9E9,9E9,9E9,9E9,9E9]];
    CONST robtarget p526:=[[463.49,37.11,0],[0,0,1,0],[-1,0,-1,0],[9E9,9E9,9E9,9E9,9E9,9E9]];
    CONST robtarget p527:=[[468.09,37.11,0],[0,0,1,0],[-1,0,-1,0],[9E9,9E9,9E9,9E9,9E9,9E9]];

    PROC DrawText()
        ! Draw text: ZignalMeister 2000

        ! Path 1/26
        ! Move to start of path (pen up)
        MoveL Offs(p0,0,0,10.0),v100,z10,tool0\WObj:=wobj0;
        ! Lower pen
        MoveL p0,v50,fine,tool0\WObj:=wobj0;
        ! Draw path
        MoveL p1,v100,z1,tool0\WObj:=wobj0;
        MoveL p2,v100,z1,tool0\WObj:=wobj0;
        MoveL p3,v100,z1,tool0\WObj:=wobj0;
        MoveL p4,v100,z1,tool0\WObj:=wobj0;
        MoveL p5,v100,z1,tool0\WObj:=wobj0;
        MoveL p6,v100,z1,tool0\WObj:=wobj0;
        MoveL p7,v100,z1,tool0\WObj:=wobj0;
        MoveL p8,v100,z1,tool0\WObj:=wobj0;
        MoveL p9,v100,z1,tool0\WObj:=wobj0;
        MoveL p10,v50,fine,tool0\WObj:=wobj0;
        ! Lift pen
        MoveL Offs(p10,0,0,10.0),v50,z10,tool0\WObj:=wobj0;

        ! Path 2/26
        ! Move to start of path (pen up)
        MoveL Offs(p11,0,0,10.0),v100,z10,tool0\WObj:=wobj0;
        ! Lower pen
        MoveL p11,v50,fine,tool0\WObj:=wobj0;
        ! Draw path
        MoveL p12,v100,z1,tool0\WObj:=wobj0;
        MoveL p13,v100,z1,tool0\WObj:=wobj0;
        MoveL p14,v100,z1,tool0\WObj:=wobj0;
        MoveL p15,v50,fine,tool0\WObj:=wobj0;
        ! Lift pen
        MoveL Offs(p15,0,0,10.0),v50,z10,tool0\WObj:=wobj0;

        ! Path 3/26
        ! Move to start of path (pen up)
        MoveL Offs(p16,0,0,10.0),v100,z10,tool0\WObj:=wobj0;
        ! Lower pen
        MoveL p16,v50,fine,tool0\WObj:=wobj0;
        ! Draw path
        MoveL p17,v100,z1,tool0\WObj:=wobj0;
        MoveL p18,v100,z1,tool0\WObj:=wobj0;
        MoveL p19,v100,z1,tool0\WObj:=wobj0;
        MoveL p20,v50,fine,tool0\WObj:=wobj0;
        ! Lift pen
        MoveL Offs(p20,0,0,10.0),v50,z10,tool0\WObj:=wobj0;

        ! Path 4/26
        ! Move to start of path (pen up)
        MoveL Offs(p21,0,0,10.0),v100,z10,tool0\WObj:=wobj0;
        ! Lower pen
        MoveL p21,v50,fine,tool0\WObj:=wobj0;
        ! Draw path
        MoveL p22,v100,z1,tool0\WObj:=wobj0;
        MoveL p23,v100,z1,tool0\WObj:=wobj0;
        MoveL p24,v100,z1,tool0\WObj:=wobj0;
        MoveL p25,v100,z1,tool0\WObj:=wobj0;
        MoveL p26,v100,z1,tool0\WObj:=wobj0;
        MoveL p27,v100,z1,tool0\WObj:=wobj0;
        MoveL p28,v100,z1,tool0\WObj:=wobj0;
        MoveL p29,v100,z1,tool0\WObj:=wobj0;
        MoveL p30,v100,z1,tool0\WObj:=wobj0;
        MoveL p31,v100,z1,tool0\WObj:=wobj0;
        MoveL p32,v100,z1,tool0\WObj:=wobj0;
        MoveL p33,v100,z1,tool0\WObj:=wobj0;
        MoveL p34,v100,z1,tool0\WObj:=wobj0;
        MoveL p35,v100,z1,tool0\WObj:=wobj0;
        MoveL p36,v100,z1,tool0\WObj:=wobj0;
        MoveL p37,v50,fine,tool0\WObj:=wobj0;
        ! Lift pen
        MoveL Offs(p37,0,0,10.0),v50,z10,tool0\WObj:=wobj0;

        ! Path 5/26
        ! Move to start of path (pen up)
        MoveL Offs(p38,0,0,10.0),v100,z10,tool0\WObj:=wobj0;
        ! Lower pen
        MoveL p38,v50,fine,tool0\WObj:=wobj0;
        ! Draw path
        MoveL p39,v100,z1,tool0\WObj:=wobj0;
        MoveL p40,v100,z1,tool0\WObj:=wobj0;
        MoveL p41,v100,z1,tool0\WObj:=wobj0;
        MoveL p42,v100,z1,tool0\WObj:=wobj0;
        MoveL p43,v100,z1,tool0\WObj:=wobj0;
        MoveL p44,v100,z1,tool0\WObj:=wobj0;
        MoveL p45,v100,z1,tool0\WObj:=wobj0;
        MoveL p46,v100,z1,tool0\WObj:=wobj0;
        MoveL p47,v100,z1,tool0\WObj:=wobj0;
        MoveL p48,v100,z1,tool0\WObj:=wobj0;
        MoveL p49,v100,z1,tool0\WObj:=wobj0;
        MoveL p50,v100,z1,tool0\WObj:=wobj0;
        MoveL p51,v100,z1,tool0\WObj:=wobj0;
        MoveL p52,v100,z1,tool0\WObj:=wobj0;
        MoveL p53,v100,z1,tool0\WObj:=wobj0;
        MoveL p54,v100,z1,tool0\WObj:=wobj0;
        MoveL p55,v100,z1,tool0\WObj:=wobj0;
        MoveL p56,v100,z1,tool0\WObj:=wobj0;
        MoveL p57,v100,z1,tool0\WObj:=wobj0;
        MoveL p58,v100,z1,tool0\WObj:=wobj0;
        MoveL p59,v100,z1,tool0\WObj:=wobj0;
        MoveL p60,v100,z1,tool0\WObj:=wobj0;
        MoveL p61,v100,z1,tool0\WObj:=wobj0;
        MoveL p62,v100,z1,tool0\WObj:=wobj0;
        MoveL p63,v100,z1,tool0\WObj:=wobj0;
        MoveL p64,v100,z1,tool0\WObj:=wobj0;
        MoveL p65,v100,z1,tool0\WObj:=wobj0;
        MoveL p66,v100,z1,tool0\WObj:=wobj0;
        MoveL p67,v100,z1,tool0\WObj:=wobj0;
        MoveL p68,v100,z1,tool0\WObj:=wobj0;
        MoveL p69,v100,z1,tool0\WObj:=wobj0;
        MoveL p70,v100,z1,tool0\WObj:=wobj0;
        MoveL p71,v100,z1,tool0\WObj:=wobj0;
        MoveL p72,v100,z1,tool0\WObj:=wobj0;
        MoveL p73,v100,z1,tool0\WObj:=wobj0;
        MoveL p74,v100,z1,tool0\WObj:=wobj0;
        MoveL p75,v100,z1,tool0\WObj:=wobj0;
        MoveL p76,v100,z1,tool0\WObj:=wobj0;
        MoveL p77,v50,fine,tool0\WObj:=wobj0;
        ! Lift pen
        MoveL Offs(p77,0,0,10.0),v50,z10,tool0\WObj:=wobj0;

        ! Path 6/26
        ! Move to start of path (pen up)
        MoveL Offs(p78,0,0,10.0),v100,z10,tool0\WObj:=wobj0;
        ! Lower pen
        MoveL p78,v50,fine,tool0\WObj:=wobj0;
        ! Draw path
        MoveL p79,v100,z1,tool0\WObj:=wobj0;
        MoveL p80,v100,z1,tool0\WObj:=wobj0;
        MoveL p81,v100,z1,tool0\WObj:=wobj0;
        MoveL p82,v100,z1,tool0\WObj:=wobj0;
        MoveL p83,v100,z1,tool0\WObj:=wobj0;
        MoveL p84,v100,z1,tool0\WObj:=wobj0;
        MoveL p85,v100,z1,tool0\WObj:=wobj0;
        MoveL p86,v100,z1,tool0\WObj:=wobj0;
        MoveL p87,v100,z1,tool0\WObj:=wobj0;
        MoveL p88,v100,z1,tool0\WObj:=wobj0;
        MoveL p89,v100,z1,tool0\WObj:=wobj0;
        MoveL p90,v100,z1,tool0\WObj:=wobj0;
        MoveL p91,v100,z1,tool0\WObj:=wobj0;
        MoveL p92,v100,z1,tool0\WObj:=wobj0;
        MoveL p93,v100,z1,tool0\WObj:=wobj0;
        MoveL p94,v100,z1,tool0\WObj:=wobj0;
        MoveL p95,v100,z1,tool0\WObj:=wobj0;
        MoveL p96,v100,z1,tool0\WObj:=wobj0;
        MoveL p97,v100,z1,tool0\WObj:=wobj0;
        MoveL p98,v100,z1,tool0\WObj:=wobj0;
        MoveL p99,v100,z1,tool0\WObj:=wobj0;
        MoveL p100,v100,z1,tool0\WObj:=wobj0;
        MoveL p101,v100,z1,tool0\WObj:=wobj0;
        MoveL p102,v50,fine,tool0\WObj:=wobj0;
        ! Lift pen
        MoveL Offs(p102,0,0,10.0),v50,z10,tool0\WObj:=wobj0;

        ! Path 7/26
        ! Move to start of path (pen up)
        MoveL Offs(p103,0,0,10.0),v100,z10,tool0\WObj:=wobj0;
        ! Lower pen
        MoveL p103,v50,fine,tool0\WObj:=wobj0;
        ! Draw path
        MoveL p104,v100,z1,tool0\WObj:=wobj0;
        MoveL p105,v100,z1,tool0\WObj:=wobj0;
        MoveL p106,v100,z1,tool0\WObj:=wobj0;
        MoveL p107,v100,z1,tool0\WObj:=wobj0;
        MoveL p108,v100,z1,tool0\WObj:=wobj0;
        MoveL p109,v100,z1,tool0\WObj:=wobj0;
        MoveL p110,v100,z1,tool0\WObj:=wobj0;
        MoveL p111,v100,z1,tool0\WObj:=wobj0;
        MoveL p112,v100,z1,tool0\WObj:=wobj0;
        MoveL p113,v100,z1,tool0\WObj:=wobj0;
        MoveL p114,v100,z1,tool0\WObj:=wobj0;
        MoveL p115,v100,z1,tool0\WObj:=wobj0;
        MoveL p116,v100,z1,tool0\WObj:=wobj0;
        MoveL p117,v50,fine,tool0\WObj:=wobj0;
        ! Lift pen
        MoveL Offs(p117,0,0,10.0),v50,z10,tool0\WObj:=wobj0;

        ! Path 8/26
        ! Move to start of path (pen up)
        MoveL Offs(p118,0,0,10.0),v100,z10,tool0\WObj:=wobj0;
        ! Lower pen
        MoveL p118,v50,fine,tool0\WObj:=wobj0;
        ! Draw path
        MoveL p119,v100,z1,tool0\WObj:=wobj0;
        MoveL p120,v100,z1,tool0\WObj:=wobj0;
        MoveL p121,v100,z1,tool0\WObj:=wobj0;
        MoveL p122,v100,z1,tool0\WObj:=wobj0;
        MoveL p123,v100,z1,tool0\WObj:=wobj0;
        MoveL p124,v100,z1,tool0\WObj:=wobj0;
        MoveL p125,v100,z1,tool0\WObj:=wobj0;
        MoveL p126,v100,z1,tool0\WObj:=wobj0;
        MoveL p127,v100,z1,tool0\WObj:=wobj0;
        MoveL p128,v100,z1,tool0\WObj:=wobj0;
        MoveL p129,v100,z1,tool0\WObj:=wobj0;
        MoveL p130,v100,z1,tool0\WObj:=wobj0;
        MoveL p131,v100,z1,tool0\WObj:=wobj0;
        MoveL p132,v100,z1,tool0\WObj:=wobj0;
        MoveL p133,v100,z1,tool0\WObj:=wobj0;
        MoveL p134,v100,z1,tool0\WObj:=wobj0;
        MoveL p135,v100,z1,tool0\WObj:=wobj0;
        MoveL p136,v100,z1,tool0\WObj:=wobj0;
        MoveL p137,v100,z1,tool0\WObj:=wobj0;
        MoveL p138,v100,z1,tool0\WObj:=wobj0;
        MoveL p139,v100,z1,tool0\WObj:=wobj0;
        MoveL p140,v100,z1,tool0\WObj:=wobj0;
        MoveL p141,v100,z1,tool0\WObj:=wobj0;
        MoveL p142,v100,z1,tool0\WObj:=wobj0;
        MoveL p143,v100,z1,tool0\WObj:=wobj0;
        MoveL p144,v100,z1,tool0\WObj:=wobj0;
        MoveL p145,v100,z1,tool0\WObj:=wobj0;
        MoveL p146,v100,z1,tool0\WObj:=wobj0;
        MoveL p147,v100,z1,tool0\WObj:=wobj0;
        MoveL p148,v100,z1,tool0\WObj:=wobj0;
        MoveL p149,v100,z1,tool0\WObj:=wobj0;
        MoveL p150,v100,z1,tool0\WObj:=wobj0;
        MoveL p151,v100,z1,tool0\WObj:=wobj0;
        MoveL p152,v50,fine,tool0\WObj:=wobj0;
        ! Lift pen
        MoveL Offs(p152,0,0,10.0),v50,z10,tool0\WObj:=wobj0;

        ! Path 9/26
        ! Move to start of path (pen up)
        MoveL Offs(p153,0,0,10.0),v100,z10,tool0\WObj:=wobj0;
        ! Lower pen
        MoveL p153,v50,fine,tool0\WObj:=wobj0;
        ! Draw path
        MoveL p154,v100,z1,tool0\WObj:=wobj0;
        MoveL p155,v100,z1,tool0\WObj:=wobj0;
        MoveL p156,v100,z1,tool0\WObj:=wobj0;
        MoveL p157,v50,fine,tool0\WObj:=wobj0;
        ! Lift pen
        MoveL Offs(p157,0,0,10.0),v50,z10,tool0\WObj:=wobj0;

        ! Path 10/26
        ! Move to start of path (pen up)
        MoveL Offs(p158,0,0,10.0),v100,z10,tool0\WObj:=wobj0;
        ! Lower pen
        MoveL p158,v50,fine,tool0\WObj:=wobj0;
        ! Draw path
        MoveL p159,v100,z1,tool0\WObj:=wobj0;
        MoveL p160,v100,z1,tool0\WObj:=wobj0;
        MoveL p161,v100,z1,tool0\WObj:=wobj0;
        MoveL p162,v100,z1,tool0\WObj:=wobj0;
        MoveL p163,v100,z1,tool0\WObj:=wobj0;
        MoveL p164,v100,z1,tool0\WObj:=wobj0;
        MoveL p165,v100,z1,tool0\WObj:=wobj0;
        MoveL p166,v100,z1,tool0\WObj:=wobj0;
        MoveL p167,v100,z1,tool0\WObj:=wobj0;
        MoveL p168,v100,z1,tool0\WObj:=wobj0;
        MoveL p169,v100,z1,tool0\WObj:=wobj0;
        MoveL p170,v100,z1,tool0\WObj:=wobj0;
        MoveL p171,v50,fine,tool0\WObj:=wobj0;
        ! Lift pen
        MoveL Offs(p171,0,0,10.0),v50,z10,tool0\WObj:=wobj0;

        ! Path 11/26
        ! Move to start of path (pen up)
        MoveL Offs(p172,0,0,10.0),v100,z10,tool0\WObj:=wobj0;
        ! Lower pen
        MoveL p172,v50,fine,tool0\WObj:=wobj0;
        ! Draw path
        MoveL p173,v100,z1,tool0\WObj:=wobj0;
        MoveL p174,v100,z1,tool0\WObj:=wobj0;
        MoveL p175,v100,z1,tool0\WObj:=wobj0;
        MoveL p176,v100,z1,tool0\WObj:=wobj0;
        MoveL p177,v100,z1,tool0\WObj:=wobj0;
        MoveL p178,v100,z1,tool0\WObj:=wobj0;
        MoveL p179,v100,z1,tool0\WObj:=wobj0;
        MoveL p180,v100,z1,tool0\WObj:=wobj0;
        MoveL p181,v100,z1,tool0\WObj:=wobj0;
        MoveL p182,v100,z1,tool0\WObj:=wobj0;
        MoveL p183,v100,z1,tool0\WObj:=wobj0;
        MoveL p184,v100,z1,tool0\WObj:=wobj0;
        MoveL p185,v100,z1,tool0\WObj:=wobj0;
        MoveL p186,v100,z1,tool0\WObj:=wobj0;
        MoveL p187,v100,z1,tool0\WObj:=wobj0;
        MoveL p188,v100,z1,tool0\WObj:=wobj0;
        MoveL p189,v100,z1,tool0\WObj:=wobj0;
        MoveL p190,v100,z1,tool0\WObj:=wobj0;
        MoveL p191,v100,z1,tool0\WObj:=wobj0;
        MoveL p192,v100,z1,tool0\WObj:=wobj0;
        MoveL p193,v100,z1,tool0\WObj:=wobj0;
        MoveL p194,v100,z1,tool0\WObj:=wobj0;
        MoveL p195,v100,z1,tool0\WObj:=wobj0;
        MoveL p196,v100,z1,tool0\WObj:=wobj0;
        MoveL p197,v100,z1,tool0\WObj:=wobj0;
        MoveL p198,v100,z1,tool0\WObj:=wobj0;
        MoveL p199,v100,z1,tool0\WObj:=wobj0;
        MoveL p200,v100,z1,tool0\WObj:=wobj0;
        MoveL p201,v100,z1,tool0\WObj:=wobj0;
        MoveL p202,v50,fine,tool0\WObj:=wobj0;
        ! Lift pen
        MoveL Offs(p202,0,0,10.0),v50,z10,tool0\WObj:=wobj0;

        ! Path 12/26
        ! Move to start of path (pen up)
        MoveL Offs(p203,0,0,10.0),v100,z10,tool0\WObj:=wobj0;
        ! Lower pen
        MoveL p203,v50,fine,tool0\WObj:=wobj0;
        ! Draw path
        MoveL p204,v100,z1,tool0\WObj:=wobj0;
        MoveL p205,v100,z1,tool0\WObj:=wobj0;
        MoveL p206,v100,z1,tool0\WObj:=wobj0;
        MoveL p207,v100,z1,tool0\WObj:=wobj0;
        MoveL p208,v100,z1,tool0\WObj:=wobj0;
        MoveL p209,v100,z1,tool0\WObj:=wobj0;
        MoveL p210,v100,z1,tool0\WObj:=wobj0;
        MoveL p211,v100,z1,tool0\WObj:=wobj0;
        MoveL p212,v50,fine,tool0\WObj:=wobj0;
        ! Lift pen
        MoveL Offs(p212,0,0,10.0),v50,z10,tool0\WObj:=wobj0;

        ! Path 13/26
        ! Move to start of path (pen up)
        MoveL Offs(p213,0,0,10.0),v100,z10,tool0\WObj:=wobj0;
        ! Lower pen
        MoveL p213,v50,fine,tool0\WObj:=wobj0;
        ! Draw path
        MoveL p214,v100,z1,tool0\WObj:=wobj0;
        MoveL p215,v100,z1,tool0\WObj:=wobj0;
        MoveL p216,v100,z1,tool0\WObj:=wobj0;
        MoveL p217,v50,fine,tool0\WObj:=wobj0;
        ! Lift pen
        MoveL Offs(p217,0,0,10.0),v50,z10,tool0\WObj:=wobj0;

        ! Path 14/26
        ! Move to start of path (pen up)
        MoveL Offs(p218,0,0,10.0),v100,z10,tool0\WObj:=wobj0;
        ! Lower pen
        MoveL p218,v50,fine,tool0\WObj:=wobj0;
        ! Draw path
        MoveL p219,v100,z1,tool0\WObj:=wobj0;
        MoveL p220,v100,z1,tool0\WObj:=wobj0;
        MoveL p221,v100,z1,tool0\WObj:=wobj0;
        MoveL p222,v50,fine,tool0\WObj:=wobj0;
        ! Lift pen
        MoveL Offs(p222,0,0,10.0),v50,z10,tool0\WObj:=wobj0;

        ! Path 15/26
        ! Move to start of path (pen up)
        MoveL Offs(p223,0,0,10.0),v100,z10,tool0\WObj:=wobj0;
        ! Lower pen
        MoveL p223,v50,fine,tool0\WObj:=wobj0;
        ! Draw path
        MoveL p224,v100,z1,tool0\WObj:=wobj0;
        MoveL p225,v100,z1,tool0\WObj:=wobj0;
        MoveL p226,v100,z1,tool0\WObj:=wobj0;
        MoveL p227,v100,z1,tool0\WObj:=wobj0;
        MoveL p228,v100,z1,tool0\WObj:=wobj0;
        MoveL p229,v100,z1,tool0\WObj:=wobj0;
        MoveL p230,v100,z1,tool0\WObj:=wobj0;
        MoveL p231,v100,z1,tool0\WObj:=wobj0;
        MoveL p232,v100,z1,tool0\WObj:=wobj0;
        MoveL p233,v100,z1,tool0\WObj:=wobj0;
        MoveL p234,v100,z1,tool0\WObj:=wobj0;
        MoveL p235,v100,z1,tool0\WObj:=wobj0;
        MoveL p236,v100,z1,tool0\WObj:=wobj0;
        MoveL p237,v100,z1,tool0\WObj:=wobj0;
        MoveL p238,v100,z1,tool0\WObj:=wobj0;
        MoveL p239,v100,z1,tool0\WObj:=wobj0;
        MoveL p240,v100,z1,tool0\WObj:=wobj0;
        MoveL p241,v100,z1,tool0\WObj:=wobj0;
        MoveL p242,v100,z1,tool0\WObj:=wobj0;
        MoveL p243,v100,z1,tool0\WObj:=wobj0;
        MoveL p244,v100,z1,tool0\WObj:=wobj0;
        MoveL p245,v100,z1,tool0\WObj:=wobj0;
        MoveL p246,v100,z1,tool0\WObj:=wobj0;
        MoveL p247,v100,z1,tool0\WObj:=wobj0;
        MoveL p248,v100,z1,tool0\WObj:=wobj0;
        MoveL p249,v100,z1,tool0\WObj:=wobj0;
        MoveL p250,v100,z1,tool0\WObj:=wobj0;
        MoveL p251,v100,z1,tool0\WObj:=wobj0;
        MoveL p252,v100,z1,tool0\WObj:=wobj0;
        MoveL p253,v100,z1,tool0\WObj:=wobj0;
        MoveL p254,v100,z1,tool0\WObj:=wobj0;
        MoveL p255,v100,z1,tool0\WObj:=wobj0;
        MoveL p256,v100,z1,tool0\WObj:=wobj0;
        MoveL p257,v100,z1,tool0\WObj:=wobj0;
        MoveL p258,v100,z1,tool0\WObj:=wobj0;
        MoveL p259,v100,z1,tool0\WObj:=wobj0;
        MoveL p260,v100,z1,tool0\WObj:=wobj0;
        MoveL p261,v100,z1,tool0\WObj:=wobj0;
        MoveL p262,v100,z1,tool0\WObj:=wobj0;
        MoveL p263,v100,z1,tool0\WObj:=wobj0;
        MoveL p264,v100,z1,tool0\WObj:=wobj0;
        MoveL p265,v100,z1,tool0\WObj:=wobj0;
        MoveL p266,v100,z1,tool0\WObj:=wobj0;
        MoveL p267,v100,z1,tool0\WObj:=wobj0;
        MoveL p268,v100,z1,tool0\WObj:=wobj0;
        MoveL p269,v100,z1,tool0\WObj:=wobj0;
        MoveL p270,v100,z1,tool0\WObj:=wobj0;
        MoveL p271,v100,z1,tool0\WObj:=wobj0;
        MoveL p272,v100,z1,tool0\WObj:=wobj0;
        MoveL p273,v100,z1,tool0\WObj:=wobj0;
        MoveL p274,v100,z1,tool0\WObj:=wobj0;
        MoveL p275,v50,fine,tool0\WObj:=wobj0;
        ! Lift pen
        MoveL Offs(p275,0,0,10.0),v50,z10,tool0\WObj:=wobj0;

        ! Path 16/26
        ! Move to start of path (pen up)
        MoveL Offs(p276,0,0,10.0),v100,z10,tool0\WObj:=wobj0;
        ! Lower pen
        MoveL p276,v50,fine,tool0\WObj:=wobj0;
        ! Draw path
        MoveL p277,v100,z1,tool0\WObj:=wobj0;
        MoveL p278,v100,z1,tool0\WObj:=wobj0;
        MoveL p279,v100,z1,tool0\WObj:=wobj0;
        MoveL p280,v100,z1,tool0\WObj:=wobj0;
        MoveL p281,v100,z1,tool0\WObj:=wobj0;
        MoveL p282,v100,z1,tool0\WObj:=wobj0;
        MoveL p283,v100,z1,tool0\WObj:=wobj0;
        MoveL p284,v100,z1,tool0\WObj:=wobj0;
        MoveL p285,v100,z1,tool0\WObj:=wobj0;
        MoveL p286,v100,z1,tool0\WObj:=wobj0;
        MoveL p287,v100,z1,tool0\WObj:=wobj0;
        MoveL p288,v100,z1,tool0\WObj:=wobj0;
        MoveL p289,v100,z1,tool0\WObj:=wobj0;
        MoveL p290,v100,z1,tool0\WObj:=wobj0;
        MoveL p291,v100,z1,tool0\WObj:=wobj0;
        MoveL p292,v100,z1,tool0\WObj:=wobj0;
        MoveL p293,v100,z1,tool0\WObj:=wobj0;
        MoveL p294,v100,z1,tool0\WObj:=wobj0;
        MoveL p295,v100,z1,tool0\WObj:=wobj0;
        MoveL p296,v100,z1,tool0\WObj:=wobj0;
        MoveL p297,v100,z1,tool0\WObj:=wobj0;
        MoveL p298,v50,fine,tool0\WObj:=wobj0;
        ! Lift pen
        MoveL Offs(p298,0,0,10.0),v50,z10,tool0\WObj:=wobj0;

        ! Path 17/26
        ! Move to start of path (pen up)
        MoveL Offs(p299,0,0,10.0),v100,z10,tool0\WObj:=wobj0;
        ! Lower pen
        MoveL p299,v50,fine,tool0\WObj:=wobj0;
        ! Draw path
        MoveL p300,v100,z1,tool0\WObj:=wobj0;
        MoveL p301,v100,z1,tool0\WObj:=wobj0;
        MoveL p302,v100,z1,tool0\WObj:=wobj0;
        MoveL p303,v100,z1,tool0\WObj:=wobj0;
        MoveL p304,v100,z1,tool0\WObj:=wobj0;
        MoveL p305,v100,z1,tool0\WObj:=wobj0;
        MoveL p306,v100,z1,tool0\WObj:=wobj0;
        MoveL p307,v100,z1,tool0\WObj:=wobj0;
        MoveL p308,v100,z1,tool0\WObj:=wobj0;
        MoveL p309,v100,z1,tool0\WObj:=wobj0;
        MoveL p310,v100,z1,tool0\WObj:=wobj0;
        MoveL p311,v100,z1,tool0\WObj:=wobj0;
        MoveL p312,v100,z1,tool0\WObj:=wobj0;
        MoveL p313,v100,z1,tool0\WObj:=wobj0;
        MoveL p314,v100,z1,tool0\WObj:=wobj0;
        MoveL p315,v100,z1,tool0\WObj:=wobj0;
        MoveL p316,v100,z1,tool0\WObj:=wobj0;
        MoveL p317,v100,z1,tool0\WObj:=wobj0;
        MoveL p318,v100,z1,tool0\WObj:=wobj0;
        MoveL p319,v100,z1,tool0\WObj:=wobj0;
        MoveL p320,v100,z1,tool0\WObj:=wobj0;
        MoveL p321,v100,z1,tool0\WObj:=wobj0;
        MoveL p322,v100,z1,tool0\WObj:=wobj0;
        MoveL p323,v100,z1,tool0\WObj:=wobj0;
        MoveL p324,v100,z1,tool0\WObj:=wobj0;
        MoveL p325,v100,z1,tool0\WObj:=wobj0;
        MoveL p326,v100,z1,tool0\WObj:=wobj0;
        MoveL p327,v100,z1,tool0\WObj:=wobj0;
        MoveL p328,v100,z1,tool0\WObj:=wobj0;
        MoveL p329,v50,fine,tool0\WObj:=wobj0;
        ! Lift pen
        MoveL Offs(p329,0,0,10.0),v50,z10,tool0\WObj:=wobj0;

        ! Path 18/26
        ! Move to start of path (pen up)
        MoveL Offs(p330,0,0,10.0),v100,z10,tool0\WObj:=wobj0;
        ! Lower pen
        MoveL p330,v50,fine,tool0\WObj:=wobj0;
        ! Draw path
        MoveL p331,v100,z1,tool0\WObj:=wobj0;
        MoveL p332,v100,z1,tool0\WObj:=wobj0;
        MoveL p333,v100,z1,tool0\WObj:=wobj0;
        MoveL p334,v100,z1,tool0\WObj:=wobj0;
        MoveL p335,v100,z1,tool0\WObj:=wobj0;
        MoveL p336,v100,z1,tool0\WObj:=wobj0;
        MoveL p337,v100,z1,tool0\WObj:=wobj0;
        MoveL p338,v100,z1,tool0\WObj:=wobj0;
        MoveL p339,v50,fine,tool0\WObj:=wobj0;
        ! Lift pen
        MoveL Offs(p339,0,0,10.0),v50,z10,tool0\WObj:=wobj0;

        ! Path 19/26
        ! Move to start of path (pen up)
        MoveL Offs(p340,0,0,10.0),v100,z10,tool0\WObj:=wobj0;
        ! Lower pen
        MoveL p340,v50,fine,tool0\WObj:=wobj0;
        ! Draw path
        MoveL p341,v100,z1,tool0\WObj:=wobj0;
        MoveL p342,v100,z1,tool0\WObj:=wobj0;
        MoveL p343,v100,z1,tool0\WObj:=wobj0;
        MoveL p344,v100,z1,tool0\WObj:=wobj0;
        MoveL p345,v100,z1,tool0\WObj:=wobj0;
        MoveL p346,v100,z1,tool0\WObj:=wobj0;
        MoveL p347,v100,z1,tool0\WObj:=wobj0;
        MoveL p348,v100,z1,tool0\WObj:=wobj0;
        MoveL p349,v100,z1,tool0\WObj:=wobj0;
        MoveL p350,v100,z1,tool0\WObj:=wobj0;
        MoveL p351,v100,z1,tool0\WObj:=wobj0;
        MoveL p352,v100,z1,tool0\WObj:=wobj0;
        MoveL p353,v100,z1,tool0\WObj:=wobj0;
        MoveL p354,v100,z1,tool0\WObj:=wobj0;
        MoveL p355,v100,z1,tool0\WObj:=wobj0;
        MoveL p356,v100,z1,tool0\WObj:=wobj0;
        MoveL p357,v100,z1,tool0\WObj:=wobj0;
        MoveL p358,v100,z1,tool0\WObj:=wobj0;
        MoveL p359,v100,z1,tool0\WObj:=wobj0;
        MoveL p360,v100,z1,tool0\WObj:=wobj0;
        MoveL p361,v100,z1,tool0\WObj:=wobj0;
        MoveL p362,v50,fine,tool0\WObj:=wobj0;
        ! Lift pen
        MoveL Offs(p362,0,0,10.0),v50,z10,tool0\WObj:=wobj0;

        ! Path 20/26
        ! Move to start of path (pen up)
        MoveL Offs(p363,0,0,10.0),v100,z10,tool0\WObj:=wobj0;
        ! Lower pen
        MoveL p363,v50,fine,tool0\WObj:=wobj0;
        ! Draw path
        MoveL p364,v100,z1,tool0\WObj:=wobj0;
        MoveL p365,v100,z1,tool0\WObj:=wobj0;
        MoveL p366,v100,z1,tool0\WObj:=wobj0;
        MoveL p367,v100,z1,tool0\WObj:=wobj0;
        MoveL p368,v100,z1,tool0\WObj:=wobj0;
        MoveL p369,v100,z1,tool0\WObj:=wobj0;
        MoveL p370,v100,z1,tool0\WObj:=wobj0;
        MoveL p371,v100,z1,tool0\WObj:=wobj0;
        MoveL p372,v100,z1,tool0\WObj:=wobj0;
        MoveL p373,v100,z1,tool0\WObj:=wobj0;
        MoveL p374,v100,z1,tool0\WObj:=wobj0;
        MoveL p375,v100,z1,tool0\WObj:=wobj0;
        MoveL p376,v100,z1,tool0\WObj:=wobj0;
        MoveL p377,v100,z1,tool0\WObj:=wobj0;
        MoveL p378,v100,z1,tool0\WObj:=wobj0;
        MoveL p379,v100,z1,tool0\WObj:=wobj0;
        MoveL p380,v100,z1,tool0\WObj:=wobj0;
        MoveL p381,v100,z1,tool0\WObj:=wobj0;
        MoveL p382,v100,z1,tool0\WObj:=wobj0;
        MoveL p383,v100,z1,tool0\WObj:=wobj0;
        MoveL p384,v100,z1,tool0\WObj:=wobj0;
        MoveL p385,v100,z1,tool0\WObj:=wobj0;
        MoveL p386,v100,z1,tool0\WObj:=wobj0;
        MoveL p387,v100,z1,tool0\WObj:=wobj0;
        MoveL p388,v100,z1,tool0\WObj:=wobj0;
        MoveL p389,v100,z1,tool0\WObj:=wobj0;
        MoveL p390,v100,z1,tool0\WObj:=wobj0;
        MoveL p391,v100,z1,tool0\WObj:=wobj0;
        MoveL p392,v100,z1,tool0\WObj:=wobj0;
        MoveL p393,v100,z1,tool0\WObj:=wobj0;
        MoveL p394,v100,z1,tool0\WObj:=wobj0;
        MoveL p395,v100,z1,tool0\WObj:=wobj0;
        MoveL p396,v100,z1,tool0\WObj:=wobj0;
        MoveL p397,v100,z1,tool0\WObj:=wobj0;
        MoveL p398,v100,z1,tool0\WObj:=wobj0;
        MoveL p399,v100,z1,tool0\WObj:=wobj0;
        MoveL p400,v100,z1,tool0\WObj:=wobj0;
        MoveL p401,v50,fine,tool0\WObj:=wobj0;
        ! Lift pen
        MoveL Offs(p401,0,0,10.0),v50,z10,tool0\WObj:=wobj0;

        ! Path 21/26
        ! Move to start of path (pen up)
        MoveL Offs(p402,0,0,10.0),v100,z10,tool0\WObj:=wobj0;
        ! Lower pen
        MoveL p402,v50,fine,tool0\WObj:=wobj0;
        ! Draw path
        MoveL p403,v100,z1,tool0\WObj:=wobj0;
        MoveL p404,v100,z1,tool0\WObj:=wobj0;
        MoveL p405,v100,z1,tool0\WObj:=wobj0;
        MoveL p406,v100,z1,tool0\WObj:=wobj0;
        MoveL p407,v100,z1,tool0\WObj:=wobj0;
        MoveL p408,v100,z1,tool0\WObj:=wobj0;
        MoveL p409,v100,z1,tool0\WObj:=wobj0;
        MoveL p410,v100,z1,tool0\WObj:=wobj0;
        MoveL p411,v100,z1,tool0\WObj:=wobj0;
        MoveL p412,v100,z1,tool0\WObj:=wobj0;
        MoveL p413,v100,z1,tool0\WObj:=wobj0;
        MoveL p414,v100,z1,tool0\WObj:=wobj0;
        MoveL p415,v100,z1,tool0\WObj:=wobj0;
        MoveL p416,v100,z1,tool0\WObj:=wobj0;
        MoveL p417,v100,z1,tool0\WObj:=wobj0;
        MoveL p418,v100,z1,tool0\WObj:=wobj0;
        MoveL p419,v100,z1,tool0\WObj:=wobj0;
        MoveL p420,v50,fine,tool0\WObj:=wobj0;
        ! Lift pen
        MoveL Offs(p420,0,0,10.0),v50,z10,tool0\WObj:=wobj0;

        ! Path 22/26
        ! Move to start of path (pen up)
        MoveL Offs(p421,0,0,10.0),v100,z10,tool0\WObj:=wobj0;
        ! Lower pen
        MoveL p421,v50,fine,tool0\WObj:=wobj0;
        ! Draw path
        MoveL p422,v100,z1,tool0\WObj:=wobj0;
        MoveL p423,v100,z1,tool0\WObj:=wobj0;
        MoveL p424,v100,z1,tool0\WObj:=wobj0;
        MoveL p425,v100,z1,tool0\WObj:=wobj0;
        MoveL p426,v100,z1,tool0\WObj:=wobj0;
        MoveL p427,v100,z1,tool0\WObj:=wobj0;
        MoveL p428,v100,z1,tool0\WObj:=wobj0;
        MoveL p429,v100,z1,tool0\WObj:=wobj0;
        MoveL p430,v100,z1,tool0\WObj:=wobj0;
        MoveL p431,v100,z1,tool0\WObj:=wobj0;
        MoveL p432,v100,z1,tool0\WObj:=wobj0;
        MoveL p433,v100,z1,tool0\WObj:=wobj0;
        MoveL p434,v100,z1,tool0\WObj:=wobj0;
        MoveL p435,v100,z1,tool0\WObj:=wobj0;
        MoveL p436,v100,z1,tool0\WObj:=wobj0;
        MoveL p437,v100,z1,tool0\WObj:=wobj0;
        MoveL p438,v100,z1,tool0\WObj:=wobj0;
        MoveL p439,v100,z1,tool0\WObj:=wobj0;
        MoveL p440,v100,z1,tool0\WObj:=wobj0;
        MoveL p441,v100,z1,tool0\WObj:=wobj0;
        MoveL p442,v100,z1,tool0\WObj:=wobj0;
        MoveL p443,v50,fine,tool0\WObj:=wobj0;
        ! Lift pen
        MoveL Offs(p443,0,0,10.0),v50,z10,tool0\WObj:=wobj0;

        ! Path 23/26
        ! Move to start of path (pen up)
        MoveL Offs(p444,0,0,10.0),v100,z10,tool0\WObj:=wobj0;
        ! Lower pen
        MoveL p444,v50,fine,tool0\WObj:=wobj0;
        ! Draw path
        MoveL p445,v100,z1,tool0\WObj:=wobj0;
        MoveL p446,v100,z1,tool0\WObj:=wobj0;
        MoveL p447,v100,z1,tool0\WObj:=wobj0;
        MoveL p448,v100,z1,tool0\WObj:=wobj0;
        MoveL p449,v100,z1,tool0\WObj:=wobj0;
        MoveL p450,v100,z1,tool0\WObj:=wobj0;
        MoveL p451,v100,z1,tool0\WObj:=wobj0;
        MoveL p452,v100,z1,tool0\WObj:=wobj0;
        MoveL p453,v100,z1,tool0\WObj:=wobj0;
        MoveL p454,v100,z1,tool0\WObj:=wobj0;
        MoveL p455,v100,z1,tool0\WObj:=wobj0;
        MoveL p456,v100,z1,tool0\WObj:=wobj0;
        MoveL p457,v100,z1,tool0\WObj:=wobj0;
        MoveL p458,v100,z1,tool0\WObj:=wobj0;
        MoveL p459,v100,z1,tool0\WObj:=wobj0;
        MoveL p460,v100,z1,tool0\WObj:=wobj0;
        MoveL p461,v100,z1,tool0\WObj:=wobj0;
        MoveL p462,v50,fine,tool0\WObj:=wobj0;
        ! Lift pen
        MoveL Offs(p462,0,0,10.0),v50,z10,tool0\WObj:=wobj0;

        ! Path 24/26
        ! Move to start of path (pen up)
        MoveL Offs(p463,0,0,10.0),v100,z10,tool0\WObj:=wobj0;
        ! Lower pen
        MoveL p463,v50,fine,tool0\WObj:=wobj0;
        ! Draw path
        MoveL p464,v100,z1,tool0\WObj:=wobj0;
        MoveL p465,v100,z1,tool0\WObj:=wobj0;
        MoveL p466,v100,z1,tool0\WObj:=wobj0;
        MoveL p467,v100,z1,tool0\WObj:=wobj0;
        MoveL p468,v100,z1,tool0\WObj:=wobj0;
        MoveL p469,v100,z1,tool0\WObj:=wobj0;
        MoveL p470,v100,z1,tool0\WObj:=wobj0;
        MoveL p471,v100,z1,tool0\WObj:=wobj0;
        MoveL p472,v100,z1,tool0\WObj:=wobj0;
        MoveL p473,v100,z1,tool0\WObj:=wobj0;
        MoveL p474,v100,z1,tool0\WObj:=wobj0;
        MoveL p475,v100,z1,tool0\WObj:=wobj0;
        MoveL p476,v100,z1,tool0\WObj:=wobj0;
        MoveL p477,v100,z1,tool0\WObj:=wobj0;
        MoveL p478,v100,z1,tool0\WObj:=wobj0;
        MoveL p479,v100,z1,tool0\WObj:=wobj0;
        MoveL p480,v100,z1,tool0\WObj:=wobj0;
        MoveL p481,v100,z1,tool0\WObj:=wobj0;
        MoveL p482,v100,z1,tool0\WObj:=wobj0;
        MoveL p483,v100,z1,tool0\WObj:=wobj0;
        MoveL p484,v100,z1,tool0\WObj:=wobj0;
        MoveL p485,v50,fine,tool0\WObj:=wobj0;
        ! Lift pen
        MoveL Offs(p485,0,0,10.0),v50,z10,tool0\WObj:=wobj0;

        ! Path 25/26
        ! Move to start of path (pen up)
        MoveL Offs(p486,0,0,10.0),v100,z10,tool0\WObj:=wobj0;
        ! Lower pen
        MoveL p486,v50,fine,tool0\WObj:=wobj0;
        ! Draw path
        MoveL p487,v100,z1,tool0\WObj:=wobj0;
        MoveL p488,v100,z1,tool0\WObj:=wobj0;
        MoveL p489,v100,z1,tool0\WObj:=wobj0;
        MoveL p490,v100,z1,tool0\WObj:=wobj0;
        MoveL p491,v100,z1,tool0\WObj:=wobj0;
        MoveL p492,v100,z1,tool0\WObj:=wobj0;
        MoveL p493,v100,z1,tool0\WObj:=wobj0;
        MoveL p494,v100,z1,tool0\WObj:=wobj0;
        MoveL p495,v100,z1,tool0\WObj:=wobj0;
        MoveL p496,v100,z1,tool0\WObj:=wobj0;
        MoveL p497,v100,z1,tool0\WObj:=wobj0;
        MoveL p498,v100,z1,tool0\WObj:=wobj0;
        MoveL p499,v100,z1,tool0\WObj:=wobj0;
        MoveL p500,v100,z1,tool0\WObj:=wobj0;
        MoveL p501,v100,z1,tool0\WObj:=wobj0;
        MoveL p502,v100,z1,tool0\WObj:=wobj0;
        MoveL p503,v100,z1,tool0\WObj:=wobj0;
        MoveL p504,v50,fine,tool0\WObj:=wobj0;
        ! Lift pen
        MoveL Offs(p504,0,0,10.0),v50,z10,tool0\WObj:=wobj0;

        ! Path 26/26
        ! Move to start of path (pen up)
        MoveL Offs(p505,0,0,10.0),v100,z10,tool0\WObj:=wobj0;
        ! Lower pen
        MoveL p505,v50,fine,tool0\WObj:=wobj0;
        ! Draw path
        MoveL p506,v100,z1,tool0\WObj:=wobj0;
        MoveL p507,v100,z1,tool0\WObj:=wobj0;
        MoveL p508,v100,z1,tool0\WObj:=wobj0;
        MoveL p509,v100,z1,tool0\WObj:=wobj0;
        MoveL p510,v100,z1,tool0\WObj:=wobj0;
        MoveL p511,v100,z1,tool0\WObj:=wobj0;
        MoveL p512,v100,z1,tool0\WObj:=wobj0;
        MoveL p513,v100,z1,tool0\WObj:=wobj0;
        MoveL p514,v100,z1,tool0\WObj:=wobj0;
        MoveL p515,v100,z1,tool0\WObj:=wobj0;
        MoveL p516,v100,z1,tool0\WObj:=wobj0;
        MoveL p517,v100,z1,tool0\WObj:=wobj0;
        MoveL p518,v100,z1,tool0\WObj:=wobj0;
        MoveL p519,v100,z1,tool0\WObj:=wobj0;
        MoveL p520,v100,z1,tool0\WObj:=wobj0;
        MoveL p521,v100,z1,tool0\WObj:=wobj0;
        MoveL p522,v100,z1,tool0\WObj:=wobj0;
        MoveL p523,v100,z1,tool0\WObj:=wobj0;
        MoveL p524,v100,z1,tool0\WObj:=wobj0;
        MoveL p525,v100,z1,tool0\WObj:=wobj0;
        MoveL p526,v100,z1,tool0\WObj:=wobj0;
        MoveL p527,v50,fine,tool0\WObj:=wobj0;
        ! Lift pen
        MoveL Offs(p527,0,0,10.0),v50,z10,tool0\WObj:=wobj0;

    ENDPROC
ENDMODULE
